Yaskawa INFORM job: tourneTRJ0.JBI

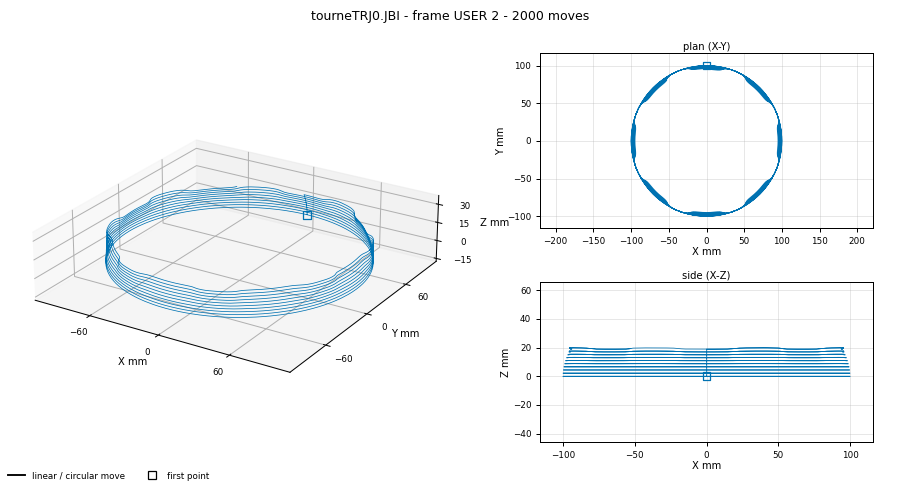
[picture p0: tool path of tourneTRJ0.JBI in frame USER 2, 2000 of 2000 moves have a stored position in this frame; points joined in program order, loops and branches not executed]
/JOB
//NAME tourneTRJ0
///FOLDERNAME DEMO
//POS
///NPOS 2000,0,2000,0,0,0
///USER 2
///TOOL 7
///POSTYPE USER
///RECTAN
///RCONF 1,0,0,0,0,0,0,0,0,0,0,0,0,0,0,0,0,0,0,0,0,0,0,0
C00000=0.000,100.000,0.000,-180.0000,-0.0000,-0.0000
C00001=5.792,99.832,0.000,-180.0000,0.0000,-3.3204
C00002=10.988,99.394,0.000,-180.0000,0.0000,-6.3084
C00003=15.564,98.781,0.000,-180.0000,0.0000,-8.9540
C00004=18.698,98.237,0.000,-180.0000,0.0000,-10.7765
C00005=20.854,97.801,0.000,-180.0000,0.0000,-12.0369
C00006=22.593,97.414,0.000,-180.0000,0.0000,-13.0576
C00007=24.351,96.990,0.000,-180.0000,0.0000,-14.0938
C00008=26.550,96.411,0.000,-180.0000,0.0000,-15.3967
C00009=29.248,95.627,0.000,-180.0000,0.0000,-17.0065
C00010=32.094,94.710,0.000,-180.0000,0.0000,-18.7198
C00011=34.739,93.772,0.000,-180.0000,0.0000,-20.3278
C00012=37.121,92.855,0.000,-180.0000,0.0000,-21.7902
C00013=39.410,91.907,0.000,-180.0000,0.0000,-23.2098
C00014=41.743,90.871,0.000,-180.0000,0.0000,-24.6724
C00015=44.276,89.664,0.000,180.0000,0.0000,-26.2801
C00016=46.937,88.300,0.000,180.0000,0.0000,-27.9935
C00017=49.400,86.946,0.000,-180.0000,0.0000,-29.6039
C00018=51.363,85.801,0.000,-180.0000,0.0000,-30.9060
C00019=52.906,84.858,0.000,-180.0000,0.0000,-31.9421
C00020=54.410,83.902,0.000,-180.0000,0.0000,-32.9632
C00021=56.242,82.685,0.000,-180.0000,0.0000,-34.2234
C00022=58.844,80.854,0.000,-180.0000,0.0000,-36.0464
C00023=62.512,78.053,0.000,-180.0000,0.0000,-38.6909
C00024=66.496,74.687,0.000,-180.0000,0.0000,-41.6796
C00025=70.711,70.711,0.000,-180.0000,0.0000,-45.0000
C00026=74.687,66.496,0.000,-180.0000,0.0000,-48.3204
C00027=78.053,62.512,0.000,-180.0000,0.0000,-51.3091
C00028=80.854,58.844,0.000,180.0000,0.0000,-53.9536
C00029=82.685,56.242,0.000,-180.0000,0.0000,-55.7766
C00030=83.902,54.410,0.000,-180.0000,0.0000,-57.0368
C00031=84.858,52.906,0.000,-180.0000,0.0000,-58.0579
C00032=85.801,51.363,0.000,-180.0000,0.0000,-59.0940
C00033=86.946,49.400,0.000,-180.0000,0.0000,-60.3961
C00034=88.300,46.937,0.000,-180.0000,0.0000,-62.0065
C00035=89.664,44.276,0.000,-180.0000,0.0000,-63.7199
C00036=90.871,41.743,0.000,-180.0000,0.0000,-65.3276
C00037=91.907,39.410,0.000,-180.0000,0.0000,-66.7902
C00038=92.855,37.121,0.000,-180.0000,0.0000,-68.2098
C00039=93.772,34.739,0.000,-180.0000,0.0000,-69.6722
C00040=94.710,32.094,0.000,-180.0000,0.0000,-71.2802
C00041=95.627,29.248,0.000,-180.0000,0.0000,-72.9935
C00042=96.411,26.550,0.000,-180.0000,0.0000,-74.6033
C00043=96.990,24.351,0.000,-180.0000,0.0000,-75.9062
C00044=97.414,22.593,0.000,-180.0000,0.0000,-76.9424
C00045=97.801,20.854,0.000,-180.0000,0.0000,-77.9631
C00046=98.237,18.698,0.000,-180.0000,0.0000,-79.2235
C00047=98.781,15.564,0.000,-180.0000,0.0000,-81.0460
C00048=99.394,10.988,0.000,-180.0000,0.0000,-83.6916
C00049=99.832,5.792,0.000,-180.0000,0.0000,-86.6796
C00050=100.000,0.000,0.000,-180.0000,0.0000,-90.0000
C00051=99.832,-5.792,0.000,-180.0000,0.0000,-93.3204
C00052=99.394,-10.988,0.000,-180.0000,0.0000,-96.3084
C00053=98.781,-15.564,0.000,-180.0000,0.0000,-98.9540
C00054=98.237,-18.698,0.000,-180.0000,0.0000,-100.7765
C00055=97.801,-20.854,0.000,-180.0000,0.0000,-102.0369
C00056=97.414,-22.593,0.000,-180.0000,0.0000,-103.0576
C00057=96.990,-24.351,0.000,-180.0000,0.0000,-104.0938
C00058=96.411,-26.550,0.000,-180.0000,0.0000,-105.3967
C00059=95.627,-29.248,0.000,-180.0000,0.0000,-107.0065
C00060=94.710,-32.094,0.000,-180.0000,0.0000,-108.7198
C00061=93.772,-34.739,0.000,-180.0000,0.0000,-110.3278
C00062=92.855,-37.121,0.000,-180.0000,0.0000,-111.7902
C00063=91.907,-39.410,0.000,-180.0000,0.0000,-113.2098
C00064=90.871,-41.743,0.000,-180.0000,0.0000,-114.6724
C00065=89.664,-44.276,0.000,-180.0000,0.0000,-116.2801
C00066=88.300,-46.937,0.000,-180.0000,0.0000,-117.9935
C00067=86.946,-49.400,0.000,-180.0000,0.0000,-119.6039
C00068=85.801,-51.363,0.000,-180.0000,0.0000,-120.9060
C00069=84.858,-52.906,0.000,-180.0000,0.0000,-121.9421
C00070=83.902,-54.410,0.000,-180.0000,0.0000,-122.9632
C00071=82.685,-56.242,0.000,-180.0000,0.0000,-124.2234
C00072=80.854,-58.844,0.000,-180.0000,0.0000,-126.0464
C00073=78.053,-62.512,0.000,-180.0000,0.0000,-128.6909
C00074=74.687,-66.496,0.000,-180.0000,0.0000,-131.6796
C00075=70.711,-70.711,0.000,-180.0000,0.0000,-135.0000
C00076=66.496,-74.687,0.000,-180.0000,0.0000,-138.3204
C00077=62.512,-78.053,0.000,-180.0000,0.0000,-141.3091
C00078=58.844,-80.854,0.000,-180.0000,0.0000,-143.9536
C00079=56.242,-82.685,0.000,-180.0000,0.0000,-145.7766
C00080=54.410,-83.902,0.000,-180.0000,0.0000,-147.0368
C00081=52.906,-84.858,0.000,-180.0000,0.0000,-148.0579
C00082=51.363,-85.801,0.000,-180.0000,0.0000,-149.0940
C00083=49.400,-86.946,0.000,180.0000,0.0000,-150.3961
C00084=46.937,-88.300,0.000,-180.0000,0.0000,-152.0065
C00085=44.276,-89.664,0.000,-180.0000,0.0000,-153.7199
C00086=41.743,-90.871,0.000,-180.0000,0.0000,-155.3276
C00087=39.410,-91.907,0.000,-180.0000,0.0000,-156.7902
C00088=37.121,-92.855,0.000,-180.0000,0.0000,-158.2098
C00089=34.739,-93.772,0.000,-180.0000,0.0000,-159.6722
C00090=32.094,-94.710,0.000,-180.0000,0.0000,-161.2802
C00091=29.248,-95.627,0.000,-180.0000,0.0000,-162.9935
C00092=26.550,-96.411,0.000,-180.0000,0.0000,-164.6033
C00093=24.351,-96.990,0.000,-180.0000,0.0000,-165.9062
C00094=22.593,-97.414,0.000,-180.0000,0.0000,-166.9424
C00095=20.854,-97.801,0.000,-180.0000,0.0000,-167.9631
C00096=18.698,-98.237,0.000,-180.0000,0.0000,-169.2235
C00097=15.564,-98.781,0.000,-180.0000,0.0000,-171.0460
C00098=10.988,-99.394,0.000,-180.0000,0.0000,-173.6916
C00099=5.792,-99.832,0.000,-180.0000,0.0000,-176.6796
C00100=0.000,-100.000,0.000,-180.0000,-0.0000,-180.0000
C00101=0.000,-100.000,0.000,-180.0000,-0.0000,-180.0000
C00102=-5.792,-99.832,0.000,180.0000,0.0000,-183.3204
C00103=-10.988,-99.394,0.000,180.0000,0.0000,-186.3084
C00104=-15.564,-98.781,0.000,180.0000,0.0000,-188.9540
C00105=-18.698,-98.237,0.000,180.0000,0.0000,-190.7765
C00106=-20.854,-97.801,0.000,180.0000,0.0000,-192.0369
C00107=-22.593,-97.414,0.000,180.0000,0.0000,-193.0576
C00108=-24.351,-96.990,0.000,180.0000,0.0000,-194.0938
C00109=-26.550,-96.411,0.000,180.0000,0.0000,-195.3967
C00110=-29.248,-95.627,0.000,180.0000,0.0000,-197.0065
C00111=-32.094,-94.710,0.000,180.0000,0.0000,-198.7198
C00112=-34.739,-93.772,0.000,180.0000,0.0000,-200.3278
C00113=-37.121,-92.855,0.000,180.0000,0.0000,-201.7902
C00114=-39.410,-91.907,0.000,180.0000,0.0000,-203.2098
C00115=-41.743,-90.871,0.000,180.0000,0.0000,-204.6724
C00116=-44.276,-89.664,0.000,180.0000,0.0000,-206.2801
C00117=-46.937,-88.300,0.000,180.0000,0.0000,-207.9935
C00118=-49.400,-86.946,0.000,180.0000,0.0000,-209.6039
C00119=-51.363,-85.801,0.000,180.0000,0.0000,-210.9060
C00120=-52.906,-84.858,0.000,180.0000,0.0000,-211.9421
C00121=-54.410,-83.902,0.000,180.0000,0.0000,-212.9632
C00122=-56.242,-82.685,0.000,180.0000,0.0000,-214.2234
C00123=-58.844,-80.854,0.000,180.0000,0.0000,-216.0464
C00124=-62.512,-78.053,0.000,180.0000,0.0000,-218.6909
C00125=-66.496,-74.687,0.000,180.0000,0.0000,-221.6796
C00126=-70.711,-70.711,0.000,180.0000,0.0000,-225.0000
C00127=-74.687,-66.496,0.000,180.0000,0.0000,-228.3204
C00128=-78.053,-62.512,0.000,180.0000,0.0000,-231.3091
C00129=-80.854,-58.844,0.000,180.0000,0.0000,-233.9536
C00130=-82.685,-56.242,0.000,180.0000,0.0000,-235.7766
C00131=-83.902,-54.410,0.000,180.0000,0.0000,-237.0368
C00132=-84.858,-52.906,0.000,180.0000,0.0000,-238.0579
C00133=-85.801,-51.363,0.000,180.0000,0.0000,-239.0940
C00134=-86.946,-49.400,0.000,180.0000,0.0000,-240.3961
C00135=-88.300,-46.937,0.000,180.0000,0.0000,-242.0065
C00136=-89.664,-44.276,0.000,180.0000,0.0000,-243.7199
C00137=-90.871,-41.743,0.000,-180.0000,0.0000,-245.3276
C00138=-91.907,-39.410,0.000,-180.0000,0.0000,-246.7902
C00139=-92.855,-37.121,0.000,180.0000,0.0000,-248.2098
C00140=-93.772,-34.739,0.000,180.0000,0.0000,-249.6722
C00141=-94.710,-32.094,0.000,-180.0000,0.0000,-251.2802
C00142=-95.627,-29.248,0.000,-180.0000,0.0000,-252.9935
C00143=-96.411,-26.550,0.000,180.0000,0.0000,-254.6033
C00144=-96.990,-24.351,0.000,180.0000,0.0000,-255.9062
C00145=-97.414,-22.593,0.000,180.0000,0.0000,-256.9424
C00146=-97.801,-20.854,0.000,180.0000,0.0000,-257.9631
C00147=-98.237,-18.698,0.000,180.0000,0.0000,-259.2235
C00148=-98.781,-15.564,0.000,180.0000,0.0000,-261.0460
C00149=-99.394,-10.988,0.000,180.0000,0.0000,-263.6916
C00150=-99.832,-5.792,0.000,180.0000,0.0000,-266.6796
C00151=-100.000,0.000,0.000,-180.0000,0.0000,-270.0000
C00152=-99.832,5.792,0.000,-180.0000,0.0000,-273.3204
C00153=-99.394,10.988,0.000,-180.0000,0.0000,-276.3084
C00154=-98.781,15.564,0.000,-180.0000,0.0000,-278.9540
C00155=-98.237,18.698,0.000,-180.0000,0.0000,-280.7765
C00156=-97.801,20.854,0.000,-180.0000,0.0000,-282.0369
C00157=-97.414,22.593,0.000,-180.0000,0.0000,-283.0576
C00158=-96.990,24.351,0.000,-180.0000,0.0000,-284.0938
C00159=-96.411,26.550,0.000,-180.0000,0.0000,-285.3967
C00160=-95.627,29.248,0.000,-180.0000,0.0000,-287.0065
C00161=-94.710,32.094,0.000,-180.0000,0.0000,-288.7198
C00162=-93.772,34.739,0.000,-180.0000,0.0000,-290.3278
C00163=-92.855,37.121,0.000,-180.0000,0.0000,-291.7902
C00164=-91.907,39.410,0.000,-180.0000,0.0000,-293.2098
C00165=-90.871,41.743,0.000,-180.0000,0.0000,-294.6724
C00166=-89.664,44.276,0.000,-180.0000,0.0000,-296.2801
C00167=-88.300,46.937,0.000,-180.0000,0.0000,-297.9935
C00168=-86.946,49.400,0.000,-180.0000,0.0000,-299.6039
C00169=-85.801,51.363,0.000,-180.0000,0.0000,-300.9060
C00170=-84.858,52.906,0.000,-180.0000,0.0000,-301.9421
C00171=-83.902,54.410,0.000,-180.0000,0.0000,-302.9632
C00172=-82.685,56.242,0.000,-180.0000,0.0000,-304.2234
C00173=-80.854,58.844,0.000,-180.0000,0.0000,-306.0464
C00174=-78.053,62.512,0.000,-180.0000,0.0000,-308.6909
C00175=-74.687,66.496,0.000,-180.0000,0.0000,-311.6796
C00176=-70.711,70.711,0.000,-180.0000,0.0000,-315.0000
C00177=-66.496,74.687,0.000,-180.0000,0.0000,-318.3204
C00178=-62.512,78.053,0.000,-180.0000,0.0000,-321.3091
C00179=-58.844,80.854,0.000,-180.0000,0.0000,-323.9536
C00180=-56.242,82.685,0.000,-180.0000,0.0000,-325.7766
C00181=-54.410,83.902,0.000,-180.0000,0.0000,-327.0368
C00182=-52.906,84.858,0.000,-180.0000,0.0000,-328.0579
C00183=-51.363,85.801,0.000,-180.0000,0.0000,-329.0940
C00184=-49.400,86.946,0.000,-180.0000,0.0000,-330.3961
C00185=-46.937,88.300,0.000,-180.0000,0.0000,-332.0065
C00186=-44.276,89.664,0.000,-180.0000,0.0000,-333.7199
C00187=-41.743,90.871,0.000,-180.0000,0.0000,-335.3276
C00188=-39.410,91.907,0.000,-180.0000,0.0000,-336.7902
C00189=-37.121,92.855,0.000,-180.0000,0.0000,-338.2098
C00190=-34.739,93.772,0.000,-180.0000,0.0000,-339.6722
C00191=-32.094,94.710,0.000,-180.0000,0.0000,-341.2802
C00192=-29.248,95.627,0.000,-180.0000,0.0000,-342.9935
C00193=-26.550,96.411,0.000,-180.0000,0.0000,-344.6033
C00194=-24.351,96.990,0.000,-180.0000,0.0000,-345.9062
C00195=-22.593,97.414,0.000,-180.0000,0.0000,-346.9424
C00196=-20.854,97.801,0.000,-180.0000,0.0000,-347.9631
C00197=-18.698,98.237,0.000,-180.0000,0.0000,-349.2235
C00198=-15.564,98.781,0.000,-180.0000,0.0000,-351.0460
C00199=-10.988,99.394,0.000,-180.0000,0.0000,-353.6916
C00200=-5.792,99.832,0.000,-180.0000,0.0000,-356.6796
C00201=0.000,100.000,0.000,-180.0000,0.0000,-360.0000
C00202=0.000,99.921,2.199,-175.9401,0.0000,-360.0000
C00203=5.785,99.754,2.199,-175.9390,-0.0000,-363.3190
C00204=10.976,99.317,2.199,-175.9440,0.0018,-366.3064
C00205=15.549,98.707,2.199,-176.1001,-0.0049,-368.9521
C00206=18.681,98.171,2.199,-176.5006,-0.0123,-370.7740
C00207=20.835,97.748,2.199,-177.0907,-0.0165,-372.0325
C00208=22.573,97.375,2.200,-177.7808,-0.0203,-373.0515
C00209=24.330,96.965,2.200,-178.4726,-0.0110,-374.0856
C00210=26.527,96.399,2.200,-179.0744,-0.0051,-375.3858
C00211=29.226,95.625,2.200,-179.5505,0.0004,-376.9948
C00212=32.077,94.713,2.200,-179.8732,-0.0006,-378.7100
C00213=34.728,93.776,2.200,-179.9819,-0.0006,-380.3211
C00214=37.118,92.856,2.200,-180.0000,0.0000,-381.7884
C00215=39.413,91.905,2.200,-180.0000,0.0000,-383.2118
C00216=41.753,90.866,2.200,-179.9796,0.0032,-384.6788
C00217=44.291,89.654,2.200,-179.8719,0.0006,-386.2904
C00218=46.951,88.283,2.200,-179.5514,0.0015,-388.0051
C00219=49.407,86.922,2.200,-179.0733,0.0071,-389.6142
C00220=51.360,85.768,2.200,-178.4728,0.0072,-390.9142
C00221=52.893,84.816,2.200,-177.7789,0.0198,-391.9485
C00222=54.385,83.851,2.199,-177.0907,0.0192,-392.9671
C00223=56.208,82.627,2.199,-176.5030,0.0134,-394.2260
C00224=58.802,80.791,2.199,-176.1018,0.0066,-396.0482
C00225=62.466,77.989,2.199,-175.9449,-0.0006,-398.6933
C00226=66.446,74.627,2.199,-175.9384,-0.0000,-401.6811
C00227=70.655,70.655,2.199,-175.9371,0.0000,-405.0000
C00228=74.627,66.446,2.199,-175.9384,0.0000,-408.3189
C00229=77.989,62.466,2.199,-175.9449,0.0006,-411.3067
C00230=80.791,58.802,2.199,-176.1018,-0.0066,-413.9518
C00231=82.627,56.208,2.199,-176.5030,-0.0134,-415.7740
C00232=83.851,54.385,2.199,-177.0907,-0.0192,-417.0329
C00233=84.816,52.893,2.200,-177.7789,-0.0198,-418.0515
C00234=85.768,51.360,2.200,-178.4728,-0.0072,-419.0858
C00235=86.922,49.407,2.200,-179.0733,-0.0071,-420.3858
C00236=88.283,46.951,2.200,-179.5514,-0.0015,-421.9949
C00237=89.654,44.291,2.200,-179.8719,-0.0006,-423.7096
C00238=90.866,41.753,2.200,-179.9796,-0.0032,-425.3212
C00239=91.905,39.413,2.200,-180.0000,0.0000,-426.7882
C00240=92.856,37.118,2.200,-180.0000,0.0000,-428.2116
C00241=93.776,34.728,2.200,-179.9819,0.0006,-429.6789
C00242=94.713,32.077,2.200,-179.8732,0.0006,-431.2900
C00243=95.625,29.226,2.200,-179.5505,-0.0004,-433.0052
C00244=96.399,26.527,2.200,-179.0744,0.0051,-434.6142
C00245=96.965,24.330,2.200,-178.4726,0.0110,-435.9144
C00246=97.375,22.573,2.200,-177.7808,0.0203,-436.9485
C00247=97.748,20.835,2.199,-177.0907,0.0165,-437.9675
C00248=98.171,18.681,2.199,-176.5006,0.0123,-439.2260
C00249=98.707,15.549,2.199,-176.1001,0.0049,-441.0479
C00250=99.317,10.976,2.199,-175.9440,-0.0018,-443.6936
C00251=99.754,5.785,2.199,-175.9390,0.0000,-446.6810
C00252=99.921,0.000,2.199,-175.9401,0.0000,-450.0000
C00253=99.754,-5.785,2.199,-175.9390,-0.0000,-453.3190
C00254=99.317,-10.976,2.199,-175.9440,0.0018,-456.3064
C00255=98.707,-15.549,2.199,-176.1001,-0.0049,-458.9521
C00256=98.171,-18.681,2.199,-176.5006,-0.0123,-460.7740
C00257=97.748,-20.835,2.199,-177.0907,-0.0165,-462.0325
C00258=97.375,-22.573,2.200,-177.7808,-0.0203,-463.0515
C00259=96.965,-24.330,2.200,-178.4726,-0.0110,-464.0856
C00260=96.399,-26.527,2.200,-179.0744,-0.0051,-465.3858
C00261=95.625,-29.226,2.200,-179.5505,0.0004,-466.9948
C00262=94.713,-32.077,2.200,-179.8732,-0.0006,-468.7100
C00263=93.776,-34.728,2.200,-179.9819,-0.0006,-470.3211
C00264=92.856,-37.118,2.200,-180.0000,0.0000,-471.7884
C00265=91.905,-39.413,2.200,-180.0000,0.0000,-473.2118
C00266=90.866,-41.753,2.200,-179.9796,0.0032,-474.6788
C00267=89.654,-44.291,2.200,-179.8719,0.0006,-476.2904
C00268=88.283,-46.951,2.200,-179.5514,0.0015,-478.0051
C00269=86.922,-49.407,2.200,-179.0733,0.0071,-479.6142
C00270=85.768,-51.360,2.200,-178.4728,0.0072,-480.9142
C00271=84.816,-52.893,2.200,-177.7789,0.0198,-481.9485
C00272=83.851,-54.385,2.199,-177.0907,0.0192,-482.9671
C00273=82.627,-56.208,2.199,-176.5030,0.0134,-484.2260
C00274=80.791,-58.802,2.199,-176.1018,0.0066,-486.0482
C00275=77.989,-62.466,2.199,-175.9449,-0.0006,-488.6933
C00276=74.627,-66.446,2.199,-175.9384,-0.0000,-491.6811
C00277=70.655,-70.655,2.199,-175.9371,-0.0000,-495.0000
C00278=66.446,-74.627,2.199,-175.9384,0.0000,-498.3189
C00279=62.466,-77.989,2.199,-175.9449,0.0006,-501.3067
C00280=58.802,-80.791,2.199,-176.1018,-0.0066,-503.9518
C00281=56.208,-82.627,2.199,-176.5030,-0.0134,-505.7740
C00282=54.385,-83.851,2.199,-177.0907,-0.0192,-507.0329
C00283=52.893,-84.816,2.200,-177.7789,-0.0198,-508.0515
C00284=51.360,-85.768,2.200,-178.4728,-0.0072,-509.0858
C00285=49.407,-86.922,2.200,-179.0733,-0.0071,-510.3858
C00286=46.951,-88.283,2.200,-179.5514,-0.0015,-511.9949
C00287=44.291,-89.654,2.200,-179.8719,-0.0006,-513.7096
C00288=41.753,-90.866,2.200,-179.9796,-0.0032,-515.3212
C00289=39.413,-91.905,2.200,-180.0000,0.0000,-516.7882
C00290=37.118,-92.856,2.200,-180.0000,0.0000,-518.2116
C00291=34.728,-93.776,2.200,-179.9819,0.0006,-519.6789
C00292=32.077,-94.713,2.200,-179.8732,0.0006,-521.2900
C00293=29.226,-95.625,2.200,-179.5505,-0.0004,-523.0052
C00294=26.527,-96.399,2.200,-179.0744,0.0051,-524.6142
C00295=24.330,-96.965,2.200,-178.4726,0.0110,-525.9144
C00296=22.573,-97.375,2.200,-177.7808,0.0203,-526.9485
C00297=20.835,-97.748,2.199,-177.0907,0.0165,-527.9675
C00298=18.681,-98.171,2.199,-176.5006,0.0123,-529.2260
C00299=15.549,-98.707,2.199,-176.1001,0.0049,-531.0479
C00300=10.976,-99.317,2.199,-175.9440,-0.0018,-533.6936
C00301=5.785,-99.754,2.199,-175.9390,0.0000,-536.6810
C00302=0.000,-99.921,2.199,-175.9401,0.0000,-540.0000
C00303=0.000,-99.921,2.199,-175.9401,0.0000,-540.0000
C00304=-5.785,-99.754,2.199,-175.9390,-0.0000,-543.3190
C00305=-10.976,-99.317,2.199,-175.9440,0.0018,-546.3064
C00306=-15.549,-98.707,2.199,-176.1001,-0.0049,-548.9521
C00307=-18.681,-98.171,2.199,-176.5006,-0.0123,-550.7740
C00308=-20.835,-97.748,2.199,-177.0907,-0.0165,-552.0325
C00309=-22.573,-97.375,2.200,-177.7808,-0.0203,-553.0515
C00310=-24.330,-96.965,2.200,-178.4726,-0.0110,-554.0856
C00311=-26.527,-96.399,2.200,-179.0744,-0.0051,-555.3858
C00312=-29.226,-95.625,2.200,-179.5505,0.0004,-556.9948
C00313=-32.077,-94.713,2.200,-179.8732,-0.0006,-558.7100
C00314=-34.728,-93.776,2.200,-179.9819,-0.0006,-560.3211
C00315=-37.118,-92.856,2.200,-180.0000,0.0000,-561.7884
C00316=-39.413,-91.905,2.200,-180.0000,0.0000,-563.2118
C00317=-41.753,-90.866,2.200,-179.9796,0.0032,-564.6788
C00318=-44.291,-89.654,2.200,-179.8719,0.0006,-566.2904
C00319=-46.951,-88.283,2.200,-179.5514,0.0015,-568.0051
C00320=-49.407,-86.922,2.200,-179.0733,0.0071,-569.6142
C00321=-51.360,-85.768,2.200,-178.4728,0.0072,-570.9142
C00322=-52.893,-84.816,2.200,-177.7789,0.0198,-571.9485
C00323=-54.385,-83.851,2.199,-177.0907,0.0192,-572.9671
C00324=-56.208,-82.627,2.199,-176.5030,0.0134,-574.2260
C00325=-58.802,-80.791,2.199,-176.1018,0.0066,-576.0482
C00326=-62.466,-77.989,2.199,-175.9449,-0.0006,-578.6933
C00327=-66.446,-74.627,2.199,-175.9384,-0.0000,-581.6811
C00328=-70.655,-70.655,2.199,-175.9371,-0.0000,-585.0000
C00329=-74.627,-66.446,2.199,-175.9384,0.0000,-588.3189
C00330=-77.989,-62.466,2.199,-175.9449,0.0006,-591.3067
C00331=-80.791,-58.802,2.199,-176.1018,-0.0066,-593.9518
C00332=-82.627,-56.208,2.199,-176.5030,-0.0134,-595.7740
C00333=-83.851,-54.385,2.199,-177.0907,-0.0192,-597.0329
C00334=-84.816,-52.893,2.200,-177.7789,-0.0198,-598.0515
C00335=-85.768,-51.360,2.200,-178.4728,-0.0072,-599.0858
C00336=-86.922,-49.407,2.200,-179.0733,-0.0071,-600.3858
C00337=-88.283,-46.951,2.200,-179.5514,-0.0015,-601.9949
C00338=-89.654,-44.291,2.200,-179.8719,-0.0006,-603.7096
C00339=-90.866,-41.753,2.200,-179.9796,-0.0032,-605.3212
C00340=-91.905,-39.413,2.200,-180.0000,0.0000,-606.7882
C00341=-92.856,-37.118,2.200,-180.0000,0.0000,-608.2116
C00342=-93.776,-34.728,2.200,-179.9819,0.0006,-609.6789
C00343=-94.713,-32.077,2.200,-179.8732,0.0006,-611.2900
C00344=-95.625,-29.226,2.200,-179.5505,-0.0004,-613.0052
C00345=-96.399,-26.527,2.200,-179.0744,0.0051,-614.6142
C00346=-96.965,-24.330,2.200,-178.4726,0.0110,-615.9144
C00347=-97.375,-22.573,2.200,-177.7808,0.0203,-616.9485
C00348=-97.748,-20.835,2.199,-177.0907,0.0165,-617.9675
C00349=-98.171,-18.681,2.199,-176.5006,0.0123,-619.2260
C00350=-98.707,-15.549,2.199,-176.1001,0.0049,-621.0479
C00351=-99.317,-10.976,2.199,-175.9440,-0.0018,-623.6936
C00352=-99.754,-5.785,2.199,-175.9390,0.0000,-626.6810
C00353=-99.921,0.000,2.199,-175.9401,0.0000,-630.0000
C00354=-99.754,5.785,2.199,-175.9390,-0.0000,-633.3190
C00355=-99.317,10.976,2.199,-175.9440,0.0018,-636.3064
C00356=-98.707,15.549,2.199,-176.1001,-0.0049,-638.9521
C00357=-98.171,18.681,2.199,-176.5006,-0.0123,-640.7740
C00358=-97.748,20.835,2.199,-177.0907,-0.0165,-642.0325
C00359=-97.375,22.573,2.200,-177.7808,-0.0203,-643.0515
C00360=-96.965,24.330,2.200,-178.4726,-0.0110,-644.0856
C00361=-96.399,26.527,2.200,-179.0744,-0.0051,-645.3858
C00362=-95.625,29.226,2.200,-179.5505,0.0004,-646.9948
C00363=-94.713,32.077,2.200,-179.8732,-0.0006,-648.7100
C00364=-93.776,34.728,2.200,-179.9819,-0.0006,-650.3211
C00365=-92.856,37.118,2.200,-180.0000,0.0000,-651.7884
C00366=-91.905,39.413,2.200,-180.0000,0.0000,-653.2118
C00367=-90.866,41.753,2.200,-179.9796,0.0032,-654.6788
C00368=-89.654,44.291,2.200,-179.8719,0.0006,-656.2904
C00369=-88.283,46.951,2.200,-179.5514,0.0015,-658.0051
C00370=-86.922,49.407,2.200,-179.0733,0.0071,-659.6142
C00371=-85.768,51.360,2.200,-178.4728,0.0072,-660.9142
C00372=-84.816,52.893,2.200,-177.7789,0.0198,-661.9485
C00373=-83.851,54.385,2.199,-177.0907,0.0192,-662.9671
C00374=-82.627,56.208,2.199,-176.5030,0.0134,-664.2260
C00375=-80.791,58.802,2.199,-176.1018,0.0066,-666.0482
C00376=-77.989,62.466,2.199,-175.9449,-0.0006,-668.6933
C00377=-74.627,66.446,2.199,-175.9384,-0.0000,-671.6811
C00378=-70.655,70.655,2.199,-175.9371,-0.0000,-675.0000
C00379=-66.446,74.627,2.199,-175.9384,0.0000,-678.3189
C00380=-62.466,77.989,2.199,-175.9449,0.0006,-681.3067
C00381=-58.802,80.791,2.199,-176.1018,-0.0066,-683.9518
C00382=-56.208,82.627,2.199,-176.5030,-0.0134,-685.7740
C00383=-54.385,83.851,2.199,-177.0907,-0.0192,-687.0329
C00384=-52.893,84.816,2.200,-177.7789,-0.0198,-688.0515
C00385=-51.360,85.768,2.200,-178.4728,-0.0072,-689.0858
C00386=-49.407,86.922,2.200,-179.0733,-0.0071,-690.3858
C00387=-46.951,88.283,2.200,-179.5514,-0.0015,-691.9949
C00388=-44.291,89.654,2.200,-179.8719,-0.0006,-693.7096
C00389=-41.753,90.866,2.200,-179.9796,-0.0032,-695.3212
C00390=-39.413,91.905,2.200,-180.0000,0.0000,-696.7882
C00391=-37.118,92.856,2.200,-180.0000,0.0000,-698.2116
C00392=-34.728,93.776,2.200,-179.9819,0.0006,-699.6789
C00393=-32.077,94.713,2.200,-179.8732,0.0006,-701.2900
C00394=-29.226,95.625,2.200,-179.5505,-0.0004,-703.0052
C00395=-26.527,96.399,2.200,-179.0744,0.0051,-704.6142
C00396=-24.330,96.965,2.200,-178.4726,0.0110,-705.9144
C00397=-22.573,97.375,2.200,-177.7808,0.0203,-706.9485
C00398=-20.835,97.748,2.199,-177.0907,0.0165,-707.9675
C00399=-18.681,98.171,2.199,-176.5006,0.0123,-709.2260
C00400=-15.549,98.707,2.199,-176.1001,0.0049,-711.0479
C00401=-10.976,99.317,2.199,-175.9440,-0.0018,-713.6936
C00402=-5.785,99.754,2.199,-175.9390,0.0000,-716.6810
C00403=0.000,99.921,2.199,-175.9401,0.0000,-720.0000
C00404=0.000,99.691,4.387,-172.1025,0.0000,-720.0000
C00405=5.764,99.524,4.387,-172.1006,0.0031,-723.3146
C00406=10.941,99.090,4.387,-172.1132,-0.0092,-726.3008
C00407=15.506,98.490,4.388,-172.4149,-0.0426,-728.9471
C00408=18.630,97.979,4.390,-173.1917,-0.1025,-730.7659
C00409=20.779,97.591,4.393,-174.3456,-0.1482,-732.0199
C00410=22.514,97.259,4.396,-175.6935,-0.1377,-733.0335
C00411=24.268,96.890,4.398,-177.0472,-0.0778,-734.0616
C00412=26.460,96.362,4.399,-178.2128,-0.0272,-735.3544
C00413=29.164,95.617,4.399,-179.1461,-0.0089,-736.9622
C00414=32.027,94.722,4.399,-179.7590,-0.0028,-738.6812
C00415=34.697,93.786,4.400,-179.9638,-0.0012,-740.3024
C00416=37.107,92.860,4.400,-179.9947,-0.0021,-741.7817
C00417=39.424,91.901,4.400,-179.9947,-0.0023,-743.2185
C00418=41.782,90.851,4.400,-179.9616,0.0013,-744.6975
C00419=44.332,89.625,4.399,-179.7566,0.0010,-746.3188
C00420=46.990,88.233,4.399,-179.1436,0.0113,-748.0383
C00421=49.428,86.848,4.399,-178.2096,0.0294,-749.6456
C00422=51.352,85.672,4.398,-177.0480,0.0751,-750.9386
C00423=52.853,84.692,4.396,-175.6950,0.1393,-751.9667
C00424=54.314,83.700,4.393,-174.3428,0.1470,-752.9801
C00425=56.108,82.455,4.390,-173.1912,0.1047,-754.2340
C00426=58.679,80.608,4.388,-172.4131,0.0429,-756.0529
C00427=62.331,77.804,4.387,-172.1130,0.0081,-758.6992
C00428=66.299,74.450,4.387,-172.0978,-0.0024,-761.6856
C00429=70.493,70.493,4.387,-172.0990,-0.0000,-765.0000
C00430=74.450,66.299,4.387,-172.0978,0.0024,-768.3144
C00431=77.804,62.331,4.387,-172.1130,-0.0081,-771.3008
C00432=80.608,58.679,4.388,-172.4131,-0.0429,-773.9471
C00433=82.455,56.108,4.390,-173.1912,-0.1047,-775.7660
C00434=83.700,54.314,4.393,-174.3428,-0.1470,-777.0199
C00435=84.692,52.853,4.396,-175.6950,-0.1393,-778.0333
C00436=85.672,51.352,4.398,-177.0480,-0.0751,-779.0614
C00437=86.848,49.428,4.399,-178.2096,-0.0294,-780.3544
C00438=88.233,46.990,4.399,-179.1436,-0.0113,-781.9617
C00439=89.625,44.332,4.399,-179.7566,-0.0010,-783.6812
C00440=90.851,41.782,4.400,-179.9616,-0.0013,-785.3025
C00441=91.901,39.424,4.400,-179.9947,0.0023,-786.7815
C00442=92.860,37.107,4.400,-179.9947,0.0021,-788.2183
C00443=93.786,34.697,4.400,-179.9638,0.0012,-789.6976
C00444=94.722,32.027,4.399,-179.7590,0.0028,-791.3188
C00445=95.617,29.164,4.399,-179.1461,0.0089,-793.0378
C00446=96.362,26.460,4.399,-178.2128,0.0272,-794.6456
C00447=96.890,24.268,4.398,-177.0472,0.0778,-795.9384
C00448=97.259,22.514,4.396,-175.6935,0.1377,-796.9665
C00449=97.591,20.779,4.393,-174.3456,0.1482,-797.9801
C00450=97.979,18.630,4.390,-173.1917,0.1025,-799.2341
C00451=98.490,15.506,4.388,-172.4149,0.0426,-801.0529
C00452=99.090,10.941,4.387,-172.1132,0.0092,-803.6992
C00453=99.524,5.764,4.387,-172.1006,-0.0031,-806.6854
C00454=99.691,0.000,4.387,-172.1025,0.0000,-810.0000
C00455=99.524,-5.764,4.387,-172.1006,0.0031,-813.3146
C00456=99.090,-10.941,4.387,-172.1132,-0.0092,-816.3008
C00457=98.490,-15.506,4.388,-172.4149,-0.0426,-818.9471
C00458=97.979,-18.630,4.390,-173.1917,-0.1025,-820.7659
C00459=97.591,-20.779,4.393,-174.3456,-0.1482,-822.0199
C00460=97.259,-22.514,4.396,-175.6935,-0.1377,-823.0335
C00461=96.890,-24.268,4.398,-177.0472,-0.0778,-824.0616
C00462=96.362,-26.460,4.399,-178.2128,-0.0272,-825.3544
C00463=95.617,-29.164,4.399,-179.1461,-0.0089,-826.9622
C00464=94.722,-32.027,4.399,-179.7590,-0.0028,-828.6812
C00465=93.786,-34.697,4.400,-179.9638,-0.0012,-830.3024
C00466=92.860,-37.107,4.400,-179.9947,-0.0021,-831.7817
C00467=91.901,-39.424,4.400,-179.9947,-0.0023,-833.2185
C00468=90.851,-41.782,4.400,-179.9616,0.0013,-834.6975
C00469=89.625,-44.332,4.399,-179.7566,0.0010,-836.3188
C00470=88.233,-46.990,4.399,-179.1436,0.0113,-838.0383
C00471=86.848,-49.428,4.399,-178.2096,0.0294,-839.6456
C00472=85.672,-51.352,4.398,-177.0480,0.0751,-840.9386
C00473=84.692,-52.853,4.396,-175.6950,0.1393,-841.9667
C00474=83.700,-54.314,4.393,-174.3428,0.1470,-842.9801
C00475=82.455,-56.108,4.390,-173.1912,0.1047,-844.2340
C00476=80.608,-58.679,4.388,-172.4131,0.0429,-846.0529
C00477=77.804,-62.331,4.387,-172.1130,0.0081,-848.6992
C00478=74.450,-66.299,4.387,-172.0978,-0.0024,-851.6856
C00479=70.493,-70.493,4.387,-172.0990,-0.0000,-855.0000
C00480=66.299,-74.450,4.387,-172.0978,0.0024,-858.3144
C00481=62.331,-77.804,4.387,-172.1130,-0.0081,-861.3008
C00482=58.679,-80.608,4.388,-172.4131,-0.0429,-863.9471
C00483=56.108,-82.455,4.390,-173.1912,-0.1047,-865.7660
C00484=54.314,-83.700,4.393,-174.3428,-0.1470,-867.0199
C00485=52.853,-84.692,4.396,-175.6950,-0.1393,-868.0333
C00486=51.352,-85.672,4.398,-177.0480,-0.0751,-869.0614
C00487=49.428,-86.848,4.399,-178.2096,-0.0294,-870.3544
C00488=46.990,-88.233,4.399,-179.1436,-0.0113,-871.9617
C00489=44.332,-89.625,4.399,-179.7566,-0.0010,-873.6812
C00490=41.782,-90.851,4.400,-179.9616,-0.0013,-875.3025
C00491=39.424,-91.901,4.400,-179.9947,0.0023,-876.7815
C00492=37.107,-92.860,4.400,-179.9947,0.0021,-878.2183
C00493=34.697,-93.786,4.400,-179.9638,0.0012,-879.6976
C00494=32.027,-94.722,4.399,-179.7590,0.0028,-881.3188
C00495=29.164,-95.617,4.399,-179.1461,0.0089,-883.0378
C00496=26.460,-96.362,4.399,-178.2128,0.0272,-884.6456
C00497=24.268,-96.890,4.398,-177.0472,0.0778,-885.9384
C00498=22.514,-97.259,4.396,-175.6935,0.1377,-886.9665
C00499=20.779,-97.591,4.393,-174.3456,0.1482,-887.9801
C00500=18.630,-97.979,4.390,-173.1917,0.1025,-889.2341
C00501=15.506,-98.490,4.388,-172.4149,0.0426,-891.0529
C00502=10.941,-99.090,4.387,-172.1132,0.0092,-893.6992
C00503=5.764,-99.524,4.387,-172.1006,-0.0031,-896.6854
C00504=0.000,-99.691,4.387,-172.1025,0.0000,-900.0000
C00505=0.000,-99.691,4.387,-172.1025,0.0000,-900.0000
C00506=-5.764,-99.524,4.387,-172.1006,0.0031,-903.3146
C00507=-10.941,-99.090,4.387,-172.1132,-0.0092,-906.3008
C00508=-15.506,-98.490,4.388,-172.4149,-0.0426,-908.9471
C00509=-18.630,-97.979,4.390,-173.1917,-0.1025,-910.7659
C00510=-20.779,-97.591,4.393,-174.3456,-0.1482,-912.0199
C00511=-22.514,-97.259,4.396,-175.6935,-0.1377,-913.0335
C00512=-24.268,-96.890,4.398,-177.0472,-0.0778,-914.0616
C00513=-26.460,-96.362,4.399,-178.2128,-0.0272,-915.3544
C00514=-29.164,-95.617,4.399,-179.1461,-0.0089,-916.9622
C00515=-32.027,-94.722,4.399,-179.7590,-0.0028,-918.6812
C00516=-34.697,-93.786,4.400,-179.9638,-0.0012,-920.3024
C00517=-37.107,-92.860,4.400,-179.9947,-0.0021,-921.7817
C00518=-39.424,-91.901,4.400,-179.9947,-0.0023,-923.2185
C00519=-41.782,-90.851,4.400,-179.9616,0.0013,-924.6975
C00520=-44.332,-89.625,4.399,-179.7566,0.0010,-926.3188
C00521=-46.990,-88.233,4.399,-179.1436,0.0113,-928.0383
C00522=-49.428,-86.848,4.399,-178.2096,0.0294,-929.6456
C00523=-51.352,-85.672,4.398,-177.0480,0.0751,-930.9386
C00524=-52.853,-84.692,4.396,-175.6950,0.1393,-931.9667
C00525=-54.314,-83.700,4.393,-174.3428,0.1470,-932.9801
C00526=-56.108,-82.455,4.390,-173.1912,0.1047,-934.2340
C00527=-58.679,-80.608,4.388,-172.4131,0.0429,-936.0529
C00528=-62.331,-77.804,4.387,-172.1130,0.0081,-938.6992
C00529=-66.299,-74.450,4.387,-172.0978,-0.0024,-941.6856
C00530=-70.493,-70.493,4.387,-172.0990,-0.0000,-945.0000
C00531=-74.450,-66.299,4.387,-172.0978,0.0024,-948.3144
C00532=-77.804,-62.331,4.387,-172.1130,-0.0081,-951.3008
C00533=-80.608,-58.679,4.388,-172.4131,-0.0429,-953.9471
C00534=-82.455,-56.108,4.390,-173.1912,-0.1047,-955.7660
C00535=-83.700,-54.314,4.393,-174.3428,-0.1470,-957.0199
C00536=-84.692,-52.853,4.396,-175.6950,-0.1393,-958.0333
C00537=-85.672,-51.352,4.398,-177.0480,-0.0751,-959.0614
C00538=-86.848,-49.428,4.399,-178.2096,-0.0294,-960.3544
C00539=-88.233,-46.990,4.399,-179.1436,-0.0113,-961.9617
C00540=-89.625,-44.332,4.399,-179.7566,-0.0010,-963.6812
C00541=-90.851,-41.782,4.400,-179.9616,-0.0013,-965.3025
C00542=-91.901,-39.424,4.400,-179.9947,0.0023,-966.7815
C00543=-92.860,-37.107,4.400,-179.9947,0.0021,-968.2183
C00544=-93.786,-34.697,4.400,-179.9638,0.0012,-969.6976
C00545=-94.722,-32.027,4.399,-179.7590,0.0028,-971.3188
C00546=-95.617,-29.164,4.399,-179.1461,0.0089,-973.0378
C00547=-96.362,-26.460,4.399,-178.2128,0.0272,-974.6456
C00548=-96.890,-24.268,4.398,-177.0472,0.0778,-975.9384
C00549=-97.259,-22.514,4.396,-175.6935,0.1377,-976.9665
C00550=-97.591,-20.779,4.393,-174.3456,0.1482,-977.9801
C00551=-97.979,-18.630,4.390,-173.1917,0.1025,-979.2341
C00552=-98.490,-15.506,4.388,-172.4149,0.0426,-981.0529
C00553=-99.090,-10.941,4.387,-172.1132,0.0092,-983.6992
C00554=-99.524,-5.764,4.387,-172.1006,-0.0031,-986.6854
C00555=-99.691,0.000,4.387,-172.1025,-0.0000,-990.0000
C00556=-99.524,5.764,4.387,-172.1006,0.0031,-993.3146
C00557=-99.090,10.941,4.387,-172.1132,-0.0092,-996.3008
C00558=-98.490,15.506,4.388,-172.4149,-0.0426,-998.9471
C00559=-97.979,18.630,4.390,-173.1917,-0.1025,-1000.7659
C00560=-97.591,20.779,4.393,-174.3456,-0.1482,-1002.0199
C00561=-97.259,22.514,4.396,-175.6935,-0.1377,-1003.0335
C00562=-96.890,24.268,4.398,-177.0472,-0.0778,-1004.0616
C00563=-96.362,26.460,4.399,-178.2128,-0.0272,-1005.3544
C00564=-95.617,29.164,4.399,-179.1461,-0.0089,-1006.9622
C00565=-94.722,32.027,4.399,-179.7590,-0.0028,-1008.6812
C00566=-93.786,34.697,4.400,-179.9638,-0.0012,-1010.3024
C00567=-92.860,37.107,4.400,-179.9947,-0.0021,-1011.7817
C00568=-91.901,39.424,4.400,-179.9947,-0.0023,-1013.2185
C00569=-90.851,41.782,4.400,-179.9616,0.0013,-1014.6975
C00570=-89.625,44.332,4.399,-179.7566,0.0010,-1016.3188
C00571=-88.233,46.990,4.399,-179.1436,0.0113,-1018.0383
C00572=-86.848,49.428,4.399,-178.2096,0.0294,-1019.6456
C00573=-85.672,51.352,4.398,-177.0480,0.0751,-1020.9386
C00574=-84.692,52.853,4.396,-175.6950,0.1393,-1021.9667
C00575=-83.700,54.314,4.393,-174.3428,0.1470,-1022.9801
C00576=-82.455,56.108,4.390,-173.1912,0.1047,-1024.2340
C00577=-80.608,58.679,4.388,-172.4131,0.0429,-1026.0529
C00578=-77.804,62.331,4.387,-172.1130,0.0081,-1028.6992
C00579=-74.450,66.299,4.387,-172.0978,-0.0024,-1031.6856
C00580=-70.493,70.493,4.387,-172.0990,0.0000,-1035.0000
C00581=-66.299,74.450,4.387,-172.0978,0.0024,-1038.3144
C00582=-62.331,77.804,4.387,-172.1130,-0.0081,-1041.3008
C00583=-58.679,80.608,4.388,-172.4131,-0.0429,-1043.9471
C00584=-56.108,82.455,4.390,-173.1912,-0.1047,-1045.7660
C00585=-54.314,83.700,4.393,-174.3428,-0.1470,-1047.0199
C00586=-52.853,84.692,4.396,-175.6950,-0.1393,-1048.0333
C00587=-51.352,85.672,4.398,-177.0480,-0.0751,-1049.0614
C00588=-49.428,86.848,4.399,-178.2096,-0.0294,-1050.3544
C00589=-46.990,88.233,4.399,-179.1436,-0.0113,-1051.9617
C00590=-44.332,89.625,4.399,-179.7566,-0.0010,-1053.6812
C00591=-41.782,90.851,4.400,-179.9616,-0.0013,-1055.3025
C00592=-39.424,91.901,4.400,-179.9947,0.0023,-1056.7815
C00593=-37.107,92.860,4.400,-179.9947,0.0021,-1058.2183
C00594=-34.697,93.786,4.400,-179.9638,0.0012,-1059.6976
C00595=-32.027,94.722,4.399,-179.7590,0.0028,-1061.3188
C00596=-29.164,95.617,4.399,-179.1461,0.0089,-1063.0378
C00597=-26.460,96.362,4.399,-178.2128,0.0272,-1064.6456
C00598=-24.268,96.890,4.398,-177.0472,0.0778,-1065.9384
C00599=-22.514,97.259,4.396,-175.6935,0.1377,-1066.9665
C00600=-20.779,97.591,4.393,-174.3456,0.1482,-1067.9801
C00601=-18.630,97.979,4.390,-173.1917,0.1025,-1069.2341
C00602=-15.506,98.490,4.388,-172.4149,0.0426,-1071.0529
C00603=-10.941,99.090,4.387,-172.1132,0.0092,-1073.6992
C00604=-5.764,99.524,4.387,-172.1006,-0.0031,-1076.6854
C00605=0.000,99.691,4.387,-172.1025,0.0000,-1080.0000
C00606=0.000,99.321,6.555,-168.5271,0.0000,-1080.0000
C00607=5.730,99.155,6.555,-168.5253,0.0014,-1083.3073
C00608=10.884,98.723,6.555,-168.5476,-0.0211,-1086.2913
C00609=15.437,98.140,6.558,-168.9780,-0.1303,-1088.9391
C00610=18.547,97.668,6.566,-170.1170,-0.3386,-1090.7524
C00611=20.687,97.336,6.576,-171.8150,-0.4851,-1091.9986
C00612=22.417,97.071,6.585,-173.8031,-0.4429,-1093.0036
C00613=24.167,96.770,6.592,-175.7648,-0.2484,-1094.0220
C00614=26.351,96.303,6.595,-177.4464,-0.0927,-1095.3030
C00615=29.062,95.605,6.597,-178.7866,-0.0275,-1096.9082
C00616=31.947,94.737,6.598,-179.6630,-0.0048,-1098.6350
C00617=34.646,93.803,6.599,-179.9457,-0.0017,-1100.2716
C00618=37.090,92.867,6.600,-179.9947,-0.0021,-1101.7712
C00619=39.440,91.893,6.600,-179.9947,-0.0023,-1103.2288
C00620=41.830,90.827,6.599,-179.9436,-0.0008,-1104.7282
C00621=44.399,89.579,6.598,-179.6644,0.0063,-1106.3649
C00622=47.053,88.152,6.597,-178.7893,0.0293,-1108.0920
C00623=49.464,86.729,6.595,-177.4408,0.0910,-1109.6973
C00624=51.338,85.515,6.592,-175.7651,0.2472,-1110.9780
C00625=52.788,84.491,6.585,-173.8020,0.4415,-1111.9962
C00626=54.199,83.455,6.576,-171.8109,0.4845,-1113.0013
C00627=55.947,82.176,6.566,-170.1166,0.3384,-1114.2478
C00628=58.480,80.311,6.558,-168.9774,0.1342,-1116.0610
C00629=62.112,77.504,6.555,-168.5500,0.0193,-1118.7088
C00630=66.061,74.165,6.555,-168.5237,-0.0027,-1121.6924
C00631=70.230,70.230,6.555,-168.5306,-0.0000,-1125.0000
C00632=74.165,66.061,6.555,-168.5237,0.0027,-1128.3076
C00633=77.504,62.112,6.555,-168.5500,-0.0193,-1131.2912
C00634=80.311,58.480,6.558,-168.9774,-0.1342,-1133.9390
C00635=82.176,55.947,6.566,-170.1166,-0.3384,-1135.7522
C00636=83.455,54.199,6.576,-171.8109,-0.4845,-1136.9987
C00637=84.491,52.788,6.585,-173.8020,-0.4415,-1138.0038
C00638=85.515,51.338,6.592,-175.7651,-0.2472,-1139.0220
C00639=86.729,49.464,6.595,-177.4408,-0.0910,-1140.3027
C00640=88.152,47.053,6.597,-178.7893,-0.0293,-1141.9080
C00641=89.579,44.399,6.598,-179.6644,-0.0063,-1143.6351
C00642=90.827,41.830,6.599,-179.9436,0.0008,-1145.2718
C00643=91.893,39.440,6.600,-179.9947,0.0023,-1146.7712
C00644=92.867,37.090,6.600,-179.9947,0.0021,-1148.2288
C00645=93.803,34.646,6.599,-179.9457,0.0017,-1149.7284
C00646=94.737,31.947,6.598,-179.6630,0.0048,-1151.3650
C00647=95.605,29.062,6.597,-178.7866,0.0275,-1153.0918
C00648=96.303,26.351,6.595,-177.4464,0.0927,-1154.6970
C00649=96.770,24.167,6.592,-175.7648,0.2484,-1155.9780
C00650=97.071,22.417,6.585,-173.8031,0.4429,-1156.9964
C00651=97.336,20.687,6.576,-171.8150,0.4851,-1158.0014
C00652=97.668,18.547,6.566,-170.1170,0.3386,-1159.2476
C00653=98.140,15.437,6.558,-168.9780,0.1303,-1161.0609
C00654=98.723,10.884,6.555,-168.5476,0.0211,-1163.7087
C00655=99.155,5.730,6.555,-168.5253,-0.0014,-1166.6927
C00656=99.321,0.000,6.555,-168.5271,-0.0000,-1170.0000
C00657=99.155,-5.730,6.555,-168.5253,0.0014,-1173.3073
C00658=98.723,-10.884,6.555,-168.5476,-0.0211,-1176.2913
C00659=98.140,-15.437,6.558,-168.9780,-0.1303,-1178.9391
C00660=97.668,-18.547,6.566,-170.1170,-0.3386,-1180.7524
C00661=97.336,-20.687,6.576,-171.8150,-0.4851,-1181.9986
C00662=97.071,-22.417,6.585,-173.8031,-0.4429,-1183.0036
C00663=96.770,-24.167,6.592,-175.7648,-0.2484,-1184.0220
C00664=96.303,-26.351,6.595,-177.4464,-0.0927,-1185.3030
C00665=95.605,-29.062,6.597,-178.7866,-0.0275,-1186.9082
C00666=94.737,-31.947,6.598,-179.6630,-0.0048,-1188.6350
C00667=93.803,-34.646,6.599,-179.9457,-0.0017,-1190.2716
C00668=92.867,-37.090,6.600,-179.9947,-0.0021,-1191.7712
C00669=91.893,-39.440,6.600,-179.9947,-0.0023,-1193.2288
C00670=90.827,-41.830,6.599,-179.9436,-0.0008,-1194.7282
C00671=89.579,-44.399,6.598,-179.6644,0.0063,-1196.3649
C00672=88.152,-47.053,6.597,-178.7893,0.0293,-1198.0920
C00673=86.729,-49.464,6.595,-177.4408,0.0910,-1199.6973
C00674=85.515,-51.338,6.592,-175.7651,0.2472,-1200.9780
C00675=84.491,-52.788,6.585,-173.8020,0.4415,-1201.9962
C00676=83.455,-54.199,6.576,-171.8109,0.4845,-1203.0013
C00677=82.176,-55.947,6.566,-170.1166,0.3384,-1204.2478
C00678=80.311,-58.480,6.558,-168.9774,0.1342,-1206.0610
C00679=77.504,-62.112,6.555,-168.5500,0.0193,-1208.7088
C00680=74.165,-66.061,6.555,-168.5237,-0.0027,-1211.6924
C00681=70.230,-70.230,6.555,-168.5306,0.0000,-1215.0000
C00682=66.061,-74.165,6.555,-168.5237,0.0027,-1218.3076
C00683=62.112,-77.504,6.555,-168.5500,-0.0193,-1221.2912
C00684=58.480,-80.311,6.558,-168.9774,-0.1342,-1223.9390
C00685=55.947,-82.176,6.566,-170.1166,-0.3384,-1225.7522
C00686=54.199,-83.455,6.576,-171.8109,-0.4845,-1226.9987
C00687=52.788,-84.491,6.585,-173.8020,-0.4415,-1228.0038
C00688=51.338,-85.515,6.592,-175.7651,-0.2472,-1229.0220
C00689=49.464,-86.729,6.595,-177.4408,-0.0910,-1230.3027
C00690=47.053,-88.152,6.597,-178.7893,-0.0293,-1231.9080
C00691=44.399,-89.579,6.598,-179.6644,-0.0063,-1233.6351
C00692=41.830,-90.827,6.599,-179.9436,0.0008,-1235.2718
C00693=39.440,-91.893,6.600,-179.9947,0.0023,-1236.7712
C00694=37.090,-92.867,6.600,-179.9947,0.0021,-1238.2288
C00695=34.646,-93.803,6.599,-179.9457,0.0017,-1239.7284
C00696=31.947,-94.737,6.598,-179.6630,0.0048,-1241.3650
C00697=29.062,-95.605,6.597,-178.7866,0.0275,-1243.0918
C00698=26.351,-96.303,6.595,-177.4464,0.0927,-1244.6970
C00699=24.167,-96.770,6.592,-175.7648,0.2484,-1245.9780
C00700=22.417,-97.071,6.585,-173.8031,0.4429,-1246.9964
C00701=20.687,-97.336,6.576,-171.8150,0.4851,-1248.0014
C00702=18.547,-97.668,6.566,-170.1170,0.3386,-1249.2476
C00703=15.437,-98.140,6.558,-168.9780,0.1303,-1251.0609
C00704=10.884,-98.723,6.555,-168.5476,0.0211,-1253.7087
C00705=5.730,-99.155,6.555,-168.5253,-0.0014,-1256.6927
C00706=0.000,-99.321,6.555,-168.5271,0.0000,-1260.0000
C00707=0.000,-99.321,6.555,-168.5271,0.0000,-1260.0000
C00708=-5.730,-99.155,6.555,-168.5253,0.0014,-1263.3073
C00709=-10.884,-98.723,6.555,-168.5476,-0.0211,-1266.2913
C00710=-15.437,-98.140,6.558,-168.9780,-0.1303,-1268.9391
C00711=-18.547,-97.668,6.566,-170.1170,-0.3386,-1270.7524
C00712=-20.687,-97.336,6.576,-171.8150,-0.4851,-1271.9986
C00713=-22.417,-97.071,6.585,-173.8031,-0.4429,-1273.0036
C00714=-24.167,-96.770,6.592,-175.7648,-0.2484,-1274.0220
C00715=-26.351,-96.303,6.595,-177.4464,-0.0927,-1275.3030
C00716=-29.062,-95.605,6.597,-178.7866,-0.0275,-1276.9082
C00717=-31.947,-94.737,6.598,-179.6630,-0.0048,-1278.6350
C00718=-34.646,-93.803,6.599,-179.9457,-0.0017,-1280.2716
C00719=-37.090,-92.867,6.600,-179.9947,-0.0021,-1281.7712
C00720=-39.440,-91.893,6.600,-179.9947,-0.0023,-1283.2288
C00721=-41.830,-90.827,6.599,-179.9436,-0.0008,-1284.7282
C00722=-44.399,-89.579,6.598,-179.6644,0.0063,-1286.3649
C00723=-47.053,-88.152,6.597,-178.7893,0.0293,-1288.0920
C00724=-49.464,-86.729,6.595,-177.4408,0.0910,-1289.6973
C00725=-51.338,-85.515,6.592,-175.7651,0.2472,-1290.9780
C00726=-52.788,-84.491,6.585,-173.8020,0.4415,-1291.9962
C00727=-54.199,-83.455,6.576,-171.8109,0.4845,-1293.0013
C00728=-55.947,-82.176,6.566,-170.1166,0.3384,-1294.2478
C00729=-58.480,-80.311,6.558,-168.9774,0.1342,-1296.0610
C00730=-62.112,-77.504,6.555,-168.5500,0.0193,-1298.7088
C00731=-66.061,-74.165,6.555,-168.5237,-0.0027,-1301.6924
C00732=-70.230,-70.230,6.555,-168.5306,0.0000,-1305.0000
C00733=-74.165,-66.061,6.555,-168.5237,0.0027,-1308.3076
C00734=-77.504,-62.112,6.555,-168.5500,-0.0193,-1311.2912
C00735=-80.311,-58.480,6.558,-168.9774,-0.1342,-1313.9390
C00736=-82.176,-55.947,6.566,-170.1166,-0.3384,-1315.7522
C00737=-83.455,-54.199,6.576,-171.8109,-0.4845,-1316.9987
C00738=-84.491,-52.788,6.585,-173.8020,-0.4415,-1318.0038
C00739=-85.515,-51.338,6.592,-175.7651,-0.2472,-1319.0220
C00740=-86.729,-49.464,6.595,-177.4408,-0.0910,-1320.3027
C00741=-88.152,-47.053,6.597,-178.7893,-0.0293,-1321.9080
C00742=-89.579,-44.399,6.598,-179.6644,-0.0063,-1323.6351
C00743=-90.827,-41.830,6.599,-179.9436,0.0008,-1325.2718
C00744=-91.893,-39.440,6.600,-179.9947,0.0023,-1326.7712
C00745=-92.867,-37.090,6.600,-179.9947,0.0021,-1328.2288
C00746=-93.803,-34.646,6.599,-179.9457,0.0017,-1329.7284
C00747=-94.737,-31.947,6.598,-179.6630,0.0048,-1331.3650
C00748=-95.605,-29.062,6.597,-178.7866,0.0275,-1333.0918
C00749=-96.303,-26.351,6.595,-177.4464,0.0927,-1334.6970
C00750=-96.770,-24.167,6.592,-175.7648,0.2484,-1335.9780
C00751=-97.071,-22.417,6.585,-173.8031,0.4429,-1336.9964
C00752=-97.336,-20.687,6.576,-171.8150,0.4851,-1338.0014
C00753=-97.668,-18.547,6.566,-170.1170,0.3386,-1339.2476
C00754=-98.140,-15.437,6.558,-168.9780,0.1303,-1341.0609
C00755=-98.723,-10.884,6.555,-168.5476,0.0211,-1343.7087
C00756=-99.155,-5.730,6.555,-168.5253,-0.0014,-1346.6927
C00757=-99.321,0.000,6.555,-168.5271,-0.0000,-1350.0000
C00758=-99.155,5.730,6.555,-168.5253,0.0014,-1353.3073
C00759=-98.723,10.884,6.555,-168.5476,-0.0211,-1356.2913
C00760=-98.140,15.437,6.558,-168.9780,-0.1303,-1358.9391
C00761=-97.668,18.547,6.566,-170.1170,-0.3386,-1360.7524
C00762=-97.336,20.687,6.576,-171.8150,-0.4851,-1361.9986
C00763=-97.071,22.417,6.585,-173.8031,-0.4429,-1363.0036
C00764=-96.770,24.167,6.592,-175.7648,-0.2484,-1364.0220
C00765=-96.303,26.351,6.595,-177.4464,-0.0927,-1365.3030
C00766=-95.605,29.062,6.597,-178.7866,-0.0275,-1366.9082
C00767=-94.737,31.947,6.598,-179.6630,-0.0048,-1368.6350
C00768=-93.803,34.646,6.599,-179.9457,-0.0017,-1370.2716
C00769=-92.867,37.090,6.600,-179.9947,-0.0021,-1371.7712
C00770=-91.893,39.440,6.600,-179.9947,-0.0023,-1373.2288
C00771=-90.827,41.830,6.599,-179.9436,-0.0008,-1374.7282
C00772=-89.579,44.399,6.598,-179.6644,0.0063,-1376.3649
C00773=-88.152,47.053,6.597,-178.7893,0.0293,-1378.0920
C00774=-86.729,49.464,6.595,-177.4408,0.0910,-1379.6973
C00775=-85.515,51.338,6.592,-175.7651,0.2472,-1380.9780
C00776=-84.491,52.788,6.585,-173.8020,0.4415,-1381.9962
C00777=-83.455,54.199,6.576,-171.8109,0.4845,-1383.0013
C00778=-82.176,55.947,6.566,-170.1166,0.3384,-1384.2478
C00779=-80.311,58.480,6.558,-168.9774,0.1342,-1386.0610
C00780=-77.504,62.112,6.555,-168.5500,0.0193,-1388.7088
C00781=-74.165,66.061,6.555,-168.5237,-0.0027,-1391.6924
C00782=-70.230,70.230,6.555,-168.5306,0.0000,-1395.0000
C00783=-66.061,74.165,6.555,-168.5237,0.0027,-1398.3076
C00784=-62.112,77.504,6.555,-168.5500,-0.0193,-1401.2912
C00785=-58.480,80.311,6.558,-168.9774,-0.1342,-1403.9390
C00786=-55.947,82.176,6.566,-170.1166,-0.3384,-1405.7522
C00787=-54.199,83.455,6.576,-171.8109,-0.4845,-1406.9987
C00788=-52.788,84.491,6.585,-173.8020,-0.4415,-1408.0038
C00789=-51.338,85.515,6.592,-175.7651,-0.2472,-1409.0220
C00790=-49.464,86.729,6.595,-177.4408,-0.0910,-1410.3027
C00791=-47.053,88.152,6.597,-178.7893,-0.0293,-1411.9080
C00792=-44.399,89.579,6.598,-179.6644,-0.0063,-1413.6351
C00793=-41.830,90.827,6.599,-179.9436,0.0008,-1415.2718
C00794=-39.440,91.893,6.600,-179.9947,0.0023,-1416.7712
C00795=-37.090,92.867,6.600,-179.9947,0.0021,-1418.2288
C00796=-34.646,93.803,6.599,-179.9457,0.0017,-1419.7284
C00797=-31.947,94.737,6.598,-179.6630,0.0048,-1421.3650
C00798=-29.062,95.605,6.597,-178.7866,0.0275,-1423.0918
C00799=-26.351,96.303,6.595,-177.4464,0.0927,-1424.6970
C00800=-24.167,96.770,6.592,-175.7648,0.2484,-1425.9780
C00801=-22.417,97.071,6.585,-173.8031,0.4429,-1426.9964
C00802=-20.687,97.336,6.576,-171.8150,0.4851,-1428.0014
C00803=-18.547,97.668,6.566,-170.1170,0.3386,-1429.2476
C00804=-15.437,98.140,6.558,-168.9780,0.1303,-1431.0609
C00805=-10.884,98.723,6.555,-168.5476,0.0211,-1433.7087
C00806=-5.730,99.155,6.555,-168.5253,-0.0014,-1436.6927
C00807=0.000,99.321,6.555,-168.5271,0.0000,-1440.0000
C00808=0.000,98.820,8.697,-165.2384,0.0000,-1440.0000
C00809=5.684,98.656,8.697,-165.2312,0.0081,-1443.2974
C00810=10.807,98.229,8.698,-165.2649,-0.0426,-1446.2783
C00811=15.344,97.668,8.705,-165.8135,-0.3013,-1448.9284
C00812=18.436,97.247,8.723,-167.3025,-0.7735,-1450.7347
C00813=20.563,96.991,8.745,-169.5499,-1.0965,-1451.9700
C00814=22.286,96.814,8.767,-172.1574,-0.9915,-1452.9633
C00815=24.029,96.606,8.782,-174.6676,-0.5533,-1453.9678
C00816=26.202,96.222,8.789,-176.7876,-0.2036,-1455.2327
C00817=28.922,95.588,8.792,-178.4919,-0.0612,-1456.8342
C00818=31.837,94.757,8.795,-179.5978,-0.0082,-1458.5716
C00819=34.577,93.826,8.798,-179.9329,-0.0003,-1460.2300
C00820=37.066,92.876,8.800,-179.9926,0.0032,-1461.7565
C00821=39.463,91.883,8.800,-179.9925,0.0030,-1463.2431
C00822=41.895,90.794,8.798,-179.9308,-0.0004,-1464.7700
C00823=44.491,89.515,8.795,-179.5977,0.0112,-1466.4284
C00824=47.140,88.042,8.792,-178.4936,0.0579,-1468.1658
C00825=49.511,86.567,8.789,-176.7866,0.2031,-1469.7669
C00826=51.320,85.302,8.782,-174.6675,0.5502,-1471.0323
C00827=52.699,84.217,8.767,-172.1605,0.9932,-1472.0364
C00828=54.043,83.124,8.745,-169.5494,1.0947,-1473.0299
C00829=55.728,81.800,8.723,-167.3050,0.7728,-1474.2655
C00830=58.212,79.911,8.705,-165.8138,0.2999,-1476.0719
C00831=61.817,77.101,8.698,-165.2633,0.0439,-1478.7215
C00832=65.741,73.780,8.697,-165.2319,-0.0068,-1481.7023
C00833=69.877,69.877,8.697,-165.2361,0.0000,-1485.0000
C00834=73.780,65.741,8.697,-165.2319,0.0068,-1488.2977
C00835=77.101,61.817,8.698,-165.2633,-0.0439,-1491.2785
C00836=79.911,58.212,8.705,-165.8138,-0.2999,-1493.9281
C00837=81.800,55.728,8.723,-167.3050,-0.7728,-1495.7345
C00838=83.124,54.043,8.745,-169.5494,-1.0947,-1496.9701
C00839=84.217,52.699,8.767,-172.1605,-0.9932,-1497.9636
C00840=85.302,51.320,8.782,-174.6675,-0.5502,-1498.9677
C00841=86.567,49.511,8.789,-176.7866,-0.2031,-1500.2331
C00842=88.042,47.140,8.792,-178.4936,-0.0579,-1501.8342
C00843=89.515,44.491,8.795,-179.5977,-0.0112,-1503.5716
C00844=90.794,41.895,8.798,-179.9308,0.0004,-1505.2300
C00845=91.883,39.463,8.800,-179.9925,-0.0030,-1506.7569
C00846=92.876,37.066,8.800,-179.9926,-0.0032,-1508.2435
C00847=93.826,34.577,8.798,-179.9329,0.0003,-1509.7700
C00848=94.757,31.837,8.795,-179.5978,0.0082,-1511.4284
C00849=95.588,28.922,8.792,-178.4919,0.0612,-1513.1658
C00850=96.222,26.202,8.789,-176.7876,0.2036,-1514.7673
C00851=96.606,24.029,8.782,-174.6676,0.5533,-1516.0322
C00852=96.814,22.286,8.767,-172.1574,0.9915,-1517.0367
C00853=96.991,20.563,8.745,-169.5499,1.0965,-1518.0300
C00854=97.247,18.436,8.723,-167.3025,0.7735,-1519.2653
C00855=97.668,15.344,8.705,-165.8135,0.3013,-1521.0716
C00856=98.229,10.807,8.698,-165.2649,0.0426,-1523.7217
C00857=98.656,5.684,8.697,-165.2312,-0.0081,-1526.7026
C00858=98.820,0.000,8.697,-165.2384,-0.0000,-1530.0000
C00859=98.656,-5.684,8.697,-165.2312,0.0081,-1533.2974
C00860=98.229,-10.807,8.698,-165.2649,-0.0426,-1536.2783
C00861=97.668,-15.344,8.705,-165.8135,-0.3013,-1538.9284
C00862=97.247,-18.436,8.723,-167.3025,-0.7735,-1540.7347
C00863=96.991,-20.563,8.745,-169.5499,-1.0965,-1541.9700
C00864=96.814,-22.286,8.767,-172.1574,-0.9915,-1542.9633
C00865=96.606,-24.029,8.782,-174.6676,-0.5533,-1543.9678
C00866=96.222,-26.202,8.789,-176.7876,-0.2036,-1545.2327
C00867=95.588,-28.922,8.792,-178.4919,-0.0612,-1546.8342
C00868=94.757,-31.837,8.795,-179.5978,-0.0082,-1548.5716
C00869=93.826,-34.577,8.798,-179.9329,-0.0003,-1550.2300
C00870=92.876,-37.066,8.800,-179.9926,0.0032,-1551.7565
C00871=91.883,-39.463,8.800,-179.9925,0.0030,-1553.2431
C00872=90.794,-41.895,8.798,-179.9308,-0.0004,-1554.7700
C00873=89.515,-44.491,8.795,-179.5977,0.0112,-1556.4284
C00874=88.042,-47.140,8.792,-178.4936,0.0579,-1558.1658
C00875=86.567,-49.511,8.789,-176.7866,0.2031,-1559.7669
C00876=85.302,-51.320,8.782,-174.6675,0.5502,-1561.0323
C00877=84.217,-52.699,8.767,-172.1605,0.9932,-1562.0364
C00878=83.124,-54.043,8.745,-169.5494,1.0947,-1563.0299
C00879=81.800,-55.728,8.723,-167.3050,0.7728,-1564.2655
C00880=79.911,-58.212,8.705,-165.8138,0.2999,-1566.0719
C00881=77.101,-61.817,8.698,-165.2633,0.0439,-1568.7215
C00882=73.780,-65.741,8.697,-165.2319,-0.0068,-1571.7023
C00883=69.877,-69.877,8.697,-165.2361,0.0000,-1575.0000
C00884=65.741,-73.780,8.697,-165.2319,0.0068,-1578.2977
C00885=61.817,-77.101,8.698,-165.2633,-0.0439,-1581.2785
C00886=58.212,-79.911,8.705,-165.8138,-0.2999,-1583.9281
C00887=55.728,-81.800,8.723,-167.3050,-0.7728,-1585.7345
C00888=54.043,-83.124,8.745,-169.5494,-1.0947,-1586.9701
C00889=52.699,-84.217,8.767,-172.1605,-0.9932,-1587.9636
C00890=51.320,-85.302,8.782,-174.6675,-0.5502,-1588.9677
C00891=49.511,-86.567,8.789,-176.7866,-0.2031,-1590.2331
C00892=47.140,-88.042,8.792,-178.4936,-0.0579,-1591.8342
C00893=44.491,-89.515,8.795,-179.5977,-0.0112,-1593.5716
C00894=41.895,-90.794,8.798,-179.9308,0.0004,-1595.2300
C00895=39.463,-91.883,8.800,-179.9925,-0.0030,-1596.7569
C00896=37.066,-92.876,8.800,-179.9926,-0.0032,-1598.2435
C00897=34.577,-93.826,8.798,-179.9329,0.0003,-1599.7700
C00898=31.837,-94.757,8.795,-179.5978,0.0082,-1601.4284
C00899=28.922,-95.588,8.792,-178.4919,0.0612,-1603.1658
C00900=26.202,-96.222,8.789,-176.7876,0.2036,-1604.7673
C00901=24.029,-96.606,8.782,-174.6676,0.5533,-1606.0322
C00902=22.286,-96.814,8.767,-172.1574,0.9915,-1607.0367
C00903=20.563,-96.991,8.745,-169.5499,1.0965,-1608.0300
C00904=18.436,-97.247,8.723,-167.3025,0.7735,-1609.2653
C00905=15.344,-97.668,8.705,-165.8135,0.3013,-1611.0716
C00906=10.807,-98.229,8.698,-165.2649,0.0426,-1613.7217
C00907=5.684,-98.656,8.697,-165.2312,-0.0081,-1616.7026
C00908=0.000,-98.820,8.697,-165.2384,0.0000,-1620.0000
C00909=0.000,-98.820,8.697,-165.2384,0.0000,-1620.0000
C00910=-5.684,-98.656,8.697,-165.2312,0.0081,-1623.2974
C00911=-10.807,-98.229,8.698,-165.2649,-0.0426,-1626.2783
C00912=-15.344,-97.668,8.705,-165.8135,-0.3013,-1628.9284
C00913=-18.436,-97.247,8.723,-167.3025,-0.7735,-1630.7347
C00914=-20.563,-96.991,8.745,-169.5499,-1.0965,-1631.9700
C00915=-22.286,-96.814,8.767,-172.1574,-0.9915,-1632.9633
C00916=-24.029,-96.606,8.782,-174.6676,-0.5533,-1633.9678
C00917=-26.202,-96.222,8.789,-176.7876,-0.2036,-1635.2327
C00918=-28.922,-95.588,8.792,-178.4919,-0.0612,-1636.8342
C00919=-31.837,-94.757,8.795,-179.5978,-0.0082,-1638.5716
C00920=-34.577,-93.826,8.798,-179.9329,-0.0003,-1640.2300
C00921=-37.066,-92.876,8.800,-179.9926,0.0032,-1641.7565
C00922=-39.463,-91.883,8.800,-179.9925,0.0030,-1643.2431
C00923=-41.895,-90.794,8.798,-179.9308,-0.0004,-1644.7700
C00924=-44.491,-89.515,8.795,-179.5977,0.0112,-1646.4284
C00925=-47.140,-88.042,8.792,-178.4936,0.0579,-1648.1658
C00926=-49.511,-86.567,8.789,-176.7866,0.2031,-1649.7669
C00927=-51.320,-85.302,8.782,-174.6675,0.5502,-1651.0323
C00928=-52.699,-84.217,8.767,-172.1605,0.9932,-1652.0364
C00929=-54.043,-83.124,8.745,-169.5494,1.0947,-1653.0299
C00930=-55.728,-81.800,8.723,-167.3050,0.7728,-1654.2655
C00931=-58.212,-79.911,8.705,-165.8138,0.2999,-1656.0719
C00932=-61.817,-77.101,8.698,-165.2633,0.0439,-1658.7215
C00933=-65.741,-73.780,8.697,-165.2319,-0.0068,-1661.7023
C00934=-69.877,-69.877,8.697,-165.2361,0.0000,-1665.0000
C00935=-73.780,-65.741,8.697,-165.2319,0.0068,-1668.2977
C00936=-77.101,-61.817,8.698,-165.2633,-0.0439,-1671.2785
C00937=-79.911,-58.212,8.705,-165.8138,-0.2999,-1673.9281
C00938=-81.800,-55.728,8.723,-167.3050,-0.7728,-1675.7345
C00939=-83.124,-54.043,8.745,-169.5494,-1.0947,-1676.9701
C00940=-84.217,-52.699,8.767,-172.1605,-0.9932,-1677.9636
C00941=-85.302,-51.320,8.782,-174.6675,-0.5502,-1678.9677
C00942=-86.567,-49.511,8.789,-176.7866,-0.2031,-1680.2331
C00943=-88.042,-47.140,8.792,-178.4936,-0.0579,-1681.8342
C00944=-89.515,-44.491,8.795,-179.5977,-0.0112,-1683.5716
C00945=-90.794,-41.895,8.798,-179.9308,0.0004,-1685.2300
C00946=-91.883,-39.463,8.800,-179.9925,-0.0030,-1686.7569
C00947=-92.876,-37.066,8.800,-179.9926,-0.0032,-1688.2435
C00948=-93.826,-34.577,8.798,-179.9329,0.0003,-1689.7700
C00949=-94.757,-31.837,8.795,-179.5978,0.0082,-1691.4284
C00950=-95.588,-28.922,8.792,-178.4919,0.0612,-1693.1658
C00951=-96.222,-26.202,8.789,-176.7876,0.2036,-1694.7673
C00952=-96.606,-24.029,8.782,-174.6676,0.5533,-1696.0322
C00953=-96.814,-22.286,8.767,-172.1574,0.9915,-1697.0367
C00954=-96.991,-20.563,8.745,-169.5499,1.0965,-1698.0300
C00955=-97.247,-18.436,8.723,-167.3025,0.7735,-1699.2653
C00956=-97.668,-15.344,8.705,-165.8135,0.3013,-1701.0716
C00957=-98.229,-10.807,8.698,-165.2649,0.0426,-1703.7217
C00958=-98.656,-5.684,8.697,-165.2312,-0.0081,-1706.7026
C00959=-98.820,0.000,8.697,-165.2384,-0.0000,-1710.0000
C00960=-98.656,5.684,8.697,-165.2312,0.0081,-1713.2974
C00961=-98.229,10.807,8.698,-165.2649,-0.0426,-1716.2783
C00962=-97.668,15.344,8.705,-165.8135,-0.3013,-1718.9284
C00963=-97.247,18.436,8.723,-167.3025,-0.7735,-1720.7347
C00964=-96.991,20.563,8.745,-169.5499,-1.0965,-1721.9700
C00965=-96.814,22.286,8.767,-172.1574,-0.9915,-1722.9633
C00966=-96.606,24.029,8.782,-174.6676,-0.5533,-1723.9678
C00967=-96.222,26.202,8.789,-176.7876,-0.2036,-1725.2327
C00968=-95.588,28.922,8.792,-178.4919,-0.0612,-1726.8342
C00969=-94.757,31.837,8.795,-179.5978,-0.0082,-1728.5716
C00970=-93.826,34.577,8.798,-179.9329,-0.0003,-1730.2300
C00971=-92.876,37.066,8.800,-179.9926,0.0032,-1731.7565
C00972=-91.883,39.463,8.800,-179.9925,0.0030,-1733.2431
C00973=-90.794,41.895,8.798,-179.9308,-0.0004,-1734.7700
C00974=-89.515,44.491,8.795,-179.5977,0.0112,-1736.4284
C00975=-88.042,47.140,8.792,-178.4936,0.0579,-1738.1658
C00976=-86.567,49.511,8.789,-176.7866,0.2031,-1739.7669
C00977=-85.302,51.320,8.782,-174.6675,0.5502,-1741.0323
C00978=-84.217,52.699,8.767,-172.1605,0.9932,-1742.0364
C00979=-83.124,54.043,8.745,-169.5494,1.0947,-1743.0299
C00980=-81.800,55.728,8.723,-167.3050,0.7728,-1744.2655
C00981=-79.911,58.212,8.705,-165.8138,0.2999,-1746.0719
C00982=-77.101,61.817,8.698,-165.2633,0.0439,-1748.7215
C00983=-73.780,65.741,8.697,-165.2319,-0.0068,-1751.7023
C00984=-69.877,69.877,8.697,-165.2361,0.0000,-1755.0000
C00985=-65.741,73.780,8.697,-165.2319,0.0068,-1758.2977
C00986=-61.817,77.101,8.698,-165.2633,-0.0439,-1761.2785
C00987=-58.212,79.911,8.705,-165.8138,-0.2999,-1763.9281
C00988=-55.728,81.800,8.723,-167.3050,-0.7728,-1765.7345
C00989=-54.043,83.124,8.745,-169.5494,-1.0947,-1766.9701
C00990=-52.699,84.217,8.767,-172.1605,-0.9932,-1767.9636
C00991=-51.320,85.302,8.782,-174.6675,-0.5502,-1768.9677
C00992=-49.511,86.567,8.789,-176.7866,-0.2031,-1770.2331
C00993=-47.140,88.042,8.792,-178.4936,-0.0579,-1771.8342
C00994=-44.491,89.515,8.795,-179.5977,-0.0112,-1773.5716
C00995=-41.895,90.794,8.798,-179.9308,0.0004,-1775.2300
C00996=-39.463,91.883,8.800,-179.9925,-0.0030,-1776.7569
C00997=-37.066,92.876,8.800,-179.9926,-0.0032,-1778.2435
C00998=-34.577,93.826,8.798,-179.9329,0.0003,-1779.7700
C00999=-31.837,94.757,8.795,-179.5978,0.0082,-1781.4284
C01000=-28.922,95.588,8.792,-178.4919,0.0612,-1783.1658
C01001=-26.202,96.222,8.789,-176.7876,0.2036,-1784.7673
C01002=-24.029,96.606,8.782,-174.6676,0.5533,-1786.0322
C01003=-22.286,96.814,8.767,-172.1574,0.9915,-1787.0367
C01004=-20.563,96.991,8.745,-169.5499,1.0965,-1788.0300
C01005=-18.436,97.247,8.723,-167.3025,0.7735,-1789.2653
C01006=-15.344,97.668,8.705,-165.8135,0.3013,-1791.0716
C01007=-10.807,98.229,8.698,-165.2649,0.0426,-1793.7217
C01008=-5.684,98.656,8.697,-165.2312,-0.0081,-1796.7026
C01009=0.000,98.820,8.697,-165.2384,0.0000,-1800.0000
C01010=0.000,98.204,10.809,-162.2409,0.0000,-1800.0000
C01011=5.628,98.041,10.809,-162.2296,0.0065,-1803.2854
C01012=10.712,97.620,10.809,-162.2684,-0.0860,-1806.2621
C01013=15.229,97.084,10.823,-162.9320,-0.5631,-1808.9150
C01014=18.298,96.727,10.856,-164.7800,-1.4494,-1810.7121
C01015=20.409,96.562,10.898,-167.6303,-2.0251,-1811.9342
C01016=22.123,96.495,10.937,-170.8622,-1.8145,-1812.9128
C01017=23.856,96.400,10.965,-173.8063,-1.0042,-1813.8997
C01018=26.016,96.121,10.978,-176.2741,-0.3675,-1815.1448
C01019=28.748,95.567,10.985,-178.2782,-0.1051,-1816.7421
C01020=31.699,94.782,10.991,-179.5634,-0.0131,-1818.4921
C01021=34.490,93.854,10.996,-179.9202,0.0012,-1820.1777
C01022=37.037,92.887,11.000,-179.9926,0.0032,-1821.7387
C01023=39.492,91.870,11.000,-179.9925,0.0030,-1823.2613
C01024=41.977,90.753,10.996,-179.9232,0.0023,-1824.8225
C01025=44.606,89.436,10.991,-179.5644,0.0132,-1826.5076
C01026=47.248,87.904,10.985,-178.2764,0.1081,-1828.2578
C01027=49.571,86.364,10.978,-176.2728,0.3667,-1829.8549
C01028=51.296,85.034,10.965,-173.8059,1.0013,-1831.1001
C01029=52.589,83.875,10.937,-170.8611,1.8135,-1832.0874
C01030=53.849,82.711,10.898,-167.6353,2.0260,-1833.0661
C01031=55.458,81.334,10.856,-164.7794,1.4482,-1834.2883
C01032=57.880,79.417,10.823,-162.9314,0.5587,-1836.0850
C01033=61.453,76.603,10.809,-162.2669,0.0851,-1838.7375
C01034=65.346,73.305,10.809,-162.2300,-0.0070,-1841.7146
C01035=69.440,69.440,10.809,-162.2384,0.0000,-1845.0000
C01036=73.305,65.346,10.809,-162.2300,0.0070,-1848.2854
C01037=76.603,61.453,10.809,-162.2669,-0.0851,-1851.2625
C01038=79.417,57.880,10.823,-162.9314,-0.5587,-1853.9150
C01039=81.334,55.458,10.856,-164.7794,-1.4482,-1855.7117
C01040=82.711,53.849,10.898,-167.6353,-2.0260,-1856.9339
C01041=83.875,52.589,10.937,-170.8611,-1.8135,-1857.9126
C01042=85.034,51.296,10.965,-173.8059,-1.0013,-1858.8999
C01043=86.364,49.571,10.978,-176.2728,-0.3667,-1860.1451
C01044=87.904,47.248,10.985,-178.2764,-0.1081,-1861.7422
C01045=89.436,44.606,10.991,-179.5644,-0.0132,-1863.4924
C01046=90.753,41.977,10.996,-179.9232,-0.0023,-1865.1775
C01047=91.870,39.492,11.000,-179.9925,-0.0030,-1866.7387
C01048=92.887,37.037,11.000,-179.9926,-0.0032,-1868.2613
C01049=93.854,34.490,10.996,-179.9202,-0.0012,-1869.8223
C01050=94.782,31.699,10.991,-179.5634,0.0131,-1871.5079
C01051=95.567,28.748,10.985,-178.2782,0.1051,-1873.2579
C01052=96.121,26.016,10.978,-176.2741,0.3675,-1874.8552
C01053=96.400,23.856,10.965,-173.8063,1.0042,-1876.1003
C01054=96.495,22.123,10.937,-170.8622,1.8145,-1877.0872
C01055=96.562,20.409,10.898,-167.6303,2.0251,-1878.0658
C01056=96.727,18.298,10.856,-164.7800,1.4494,-1879.2879
C01057=97.084,15.229,10.823,-162.9320,0.5631,-1881.0850
C01058=97.620,10.712,10.809,-162.2684,0.0860,-1883.7379
C01059=98.041,5.628,10.809,-162.2296,-0.0065,-1886.7146
C01060=98.204,0.000,10.809,-162.2409,-0.0000,-1890.0000
C01061=98.041,-5.628,10.809,-162.2296,0.0065,-1893.2854
C01062=97.620,-10.712,10.809,-162.2684,-0.0860,-1896.2621
C01063=97.084,-15.229,10.823,-162.9320,-0.5631,-1898.9150
C01064=96.727,-18.298,10.856,-164.7800,-1.4494,-1900.7121
C01065=96.562,-20.409,10.898,-167.6303,-2.0251,-1901.9342
C01066=96.495,-22.123,10.937,-170.8622,-1.8145,-1902.9128
C01067=96.400,-23.856,10.965,-173.8063,-1.0042,-1903.8997
C01068=96.121,-26.016,10.978,-176.2741,-0.3675,-1905.1448
C01069=95.567,-28.748,10.985,-178.2782,-0.1051,-1906.7421
C01070=94.782,-31.699,10.991,-179.5634,-0.0131,-1908.4921
C01071=93.854,-34.490,10.996,-179.9202,0.0012,-1910.1777
C01072=92.887,-37.037,11.000,-179.9926,0.0032,-1911.7387
C01073=91.870,-39.492,11.000,-179.9925,0.0030,-1913.2613
C01074=90.753,-41.977,10.996,-179.9232,0.0023,-1914.8225
C01075=89.436,-44.606,10.991,-179.5644,0.0132,-1916.5076
C01076=87.904,-47.248,10.985,-178.2764,0.1081,-1918.2578
C01077=86.364,-49.571,10.978,-176.2728,0.3667,-1919.8549
C01078=85.034,-51.296,10.965,-173.8059,1.0013,-1921.1001
C01079=83.875,-52.589,10.937,-170.8611,1.8135,-1922.0874
C01080=82.711,-53.849,10.898,-167.6353,2.0260,-1923.0661
C01081=81.334,-55.458,10.856,-164.7794,1.4482,-1924.2883
C01082=79.417,-57.880,10.823,-162.9314,0.5587,-1926.0850
C01083=76.603,-61.453,10.809,-162.2669,0.0851,-1928.7375
C01084=73.305,-65.346,10.809,-162.2300,-0.0070,-1931.7146
C01085=69.440,-69.440,10.809,-162.2384,0.0000,-1935.0000
C01086=65.346,-73.305,10.809,-162.2300,0.0070,-1938.2854
C01087=61.453,-76.603,10.809,-162.2669,-0.0851,-1941.2625
C01088=57.880,-79.417,10.823,-162.9314,-0.5587,-1943.9150
C01089=55.458,-81.334,10.856,-164.7794,-1.4482,-1945.7117
C01090=53.849,-82.711,10.898,-167.6353,-2.0260,-1946.9339
C01091=52.589,-83.875,10.937,-170.8611,-1.8135,-1947.9126
C01092=51.296,-85.034,10.965,-173.8059,-1.0013,-1948.8999
C01093=49.571,-86.364,10.978,-176.2728,-0.3667,-1950.1451
C01094=47.248,-87.904,10.985,-178.2764,-0.1081,-1951.7422
C01095=44.606,-89.436,10.991,-179.5644,-0.0132,-1953.4924
C01096=41.977,-90.753,10.996,-179.9232,-0.0023,-1955.1775
C01097=39.492,-91.870,11.000,-179.9925,-0.0030,-1956.7387
C01098=37.037,-92.887,11.000,-179.9926,-0.0032,-1958.2613
C01099=34.490,-93.854,10.996,-179.9202,-0.0012,-1959.8223
C01100=31.699,-94.782,10.991,-179.5634,0.0131,-1961.5079
C01101=28.748,-95.567,10.985,-178.2782,0.1051,-1963.2579
C01102=26.016,-96.121,10.978,-176.2741,0.3675,-1964.8552
C01103=23.856,-96.400,10.965,-173.8063,1.0042,-1966.1003
C01104=22.123,-96.495,10.937,-170.8622,1.8145,-1967.0872
C01105=20.409,-96.562,10.898,-167.6303,2.0251,-1968.0658
C01106=18.298,-96.727,10.856,-164.7800,1.4494,-1969.2879
C01107=15.229,-97.084,10.823,-162.9320,0.5631,-1971.0850
C01108=10.712,-97.620,10.809,-162.2684,0.0860,-1973.7379
C01109=5.628,-98.041,10.809,-162.2296,-0.0065,-1976.7146
C01110=0.000,-98.204,10.809,-162.2409,-0.0000,-1980.0000
C01111=0.000,-98.204,10.809,-162.2409,-0.0000,-1980.0000
C01112=-5.628,-98.041,10.809,-162.2296,0.0065,-1983.2854
C01113=-10.712,-97.620,10.809,-162.2684,-0.0860,-1986.2621
C01114=-15.229,-97.084,10.823,-162.9320,-0.5631,-1988.9150
C01115=-18.298,-96.727,10.856,-164.7800,-1.4494,-1990.7121
C01116=-20.409,-96.562,10.898,-167.6303,-2.0251,-1991.9342
C01117=-22.123,-96.495,10.937,-170.8622,-1.8145,-1992.9128
C01118=-23.856,-96.400,10.965,-173.8063,-1.0042,-1993.8997
C01119=-26.016,-96.121,10.978,-176.2741,-0.3675,-1995.1448
C01120=-28.748,-95.567,10.985,-178.2782,-0.1051,-1996.7421
C01121=-31.699,-94.782,10.991,-179.5634,-0.0131,-1998.4921
C01122=-34.490,-93.854,10.996,-179.9202,0.0012,-2000.1777
C01123=-37.037,-92.887,11.000,-179.9926,0.0032,-2001.7387
C01124=-39.492,-91.870,11.000,-179.9925,0.0030,-2003.2613
C01125=-41.977,-90.753,10.996,-179.9232,0.0023,-2004.8225
C01126=-44.606,-89.436,10.991,-179.5644,0.0132,-2006.5076
C01127=-47.248,-87.904,10.985,-178.2764,0.1081,-2008.2578
C01128=-49.571,-86.364,10.978,-176.2728,0.3667,-2009.8549
C01129=-51.296,-85.034,10.965,-173.8059,1.0013,-2011.1001
C01130=-52.589,-83.875,10.937,-170.8611,1.8135,-2012.0874
C01131=-53.849,-82.711,10.898,-167.6353,2.0260,-2013.0661
C01132=-55.458,-81.334,10.856,-164.7794,1.4482,-2014.2883
C01133=-57.880,-79.417,10.823,-162.9314,0.5587,-2016.0850
C01134=-61.453,-76.603,10.809,-162.2669,0.0851,-2018.7375
C01135=-65.346,-73.305,10.809,-162.2300,-0.0070,-2021.7146
C01136=-69.440,-69.440,10.809,-162.2384,0.0000,-2025.0000
C01137=-73.305,-65.346,10.809,-162.2300,0.0070,-2028.2854
C01138=-76.603,-61.453,10.809,-162.2669,-0.0851,-2031.2625
C01139=-79.417,-57.880,10.823,-162.9314,-0.5587,-2033.9150
C01140=-81.334,-55.458,10.856,-164.7794,-1.4482,-2035.7117
C01141=-82.711,-53.849,10.898,-167.6353,-2.0260,-2036.9339
C01142=-83.875,-52.589,10.937,-170.8611,-1.8135,-2037.9126
C01143=-85.034,-51.296,10.965,-173.8059,-1.0013,-2038.8999
C01144=-86.364,-49.571,10.978,-176.2728,-0.3667,-2040.1451
C01145=-87.904,-47.248,10.985,-178.2764,-0.1081,-2041.7422
C01146=-89.436,-44.606,10.991,-179.5644,-0.0132,-2043.4924
C01147=-90.753,-41.977,10.996,-179.9232,-0.0023,-2045.1775
C01148=-91.870,-39.492,11.000,-179.9925,-0.0030,-2046.7387
C01149=-92.887,-37.037,11.000,-179.9926,-0.0032,-2048.2613
C01150=-93.854,-34.490,10.996,-179.9202,-0.0012,-2049.8223
C01151=-94.782,-31.699,10.991,-179.5634,0.0131,-2051.5079
C01152=-95.567,-28.748,10.985,-178.2782,0.1051,-2053.2579
C01153=-96.121,-26.016,10.978,-176.2741,0.3675,-2054.8552
C01154=-96.400,-23.856,10.965,-173.8063,1.0042,-2056.1003
C01155=-96.495,-22.123,10.937,-170.8622,1.8145,-2057.0872
C01156=-96.562,-20.409,10.898,-167.6303,2.0251,-2058.0658
C01157=-96.727,-18.298,10.856,-164.7800,1.4494,-2059.2879
C01158=-97.084,-15.229,10.823,-162.9320,0.5631,-2061.0850
C01159=-97.620,-10.712,10.809,-162.2684,0.0860,-2063.7379
C01160=-98.041,-5.628,10.809,-162.2296,-0.0065,-2066.7146
C01161=-98.204,0.000,10.809,-162.2409,0.0000,-2070.0000
C01162=-98.041,5.628,10.809,-162.2296,0.0065,-2073.2854
C01163=-97.620,10.712,10.809,-162.2684,-0.0860,-2076.2621
C01164=-97.084,15.229,10.823,-162.9320,-0.5631,-2078.9150
C01165=-96.727,18.298,10.856,-164.7800,-1.4494,-2080.7121
C01166=-96.562,20.409,10.898,-167.6303,-2.0251,-2081.9342
C01167=-96.495,22.123,10.937,-170.8622,-1.8145,-2082.9128
C01168=-96.400,23.856,10.965,-173.8063,-1.0042,-2083.8997
C01169=-96.121,26.016,10.978,-176.2741,-0.3675,-2085.1448
C01170=-95.567,28.748,10.985,-178.2782,-0.1051,-2086.7421
C01171=-94.782,31.699,10.991,-179.5634,-0.0131,-2088.4921
C01172=-93.854,34.490,10.996,-179.9202,0.0012,-2090.1777
C01173=-92.887,37.037,11.000,-179.9926,0.0032,-2091.7387
C01174=-91.870,39.492,11.000,-179.9925,0.0030,-2093.2613
C01175=-90.753,41.977,10.996,-179.9232,0.0023,-2094.8225
C01176=-89.436,44.606,10.991,-179.5644,0.0132,-2096.5076
C01177=-87.904,47.248,10.985,-178.2764,0.1081,-2098.2578
C01178=-86.364,49.571,10.978,-176.2728,0.3667,-2099.8549
C01179=-85.034,51.296,10.965,-173.8059,1.0013,-2101.1001
C01180=-83.875,52.589,10.937,-170.8611,1.8135,-2102.0874
C01181=-82.711,53.849,10.898,-167.6353,2.0260,-2103.0661
C01182=-81.334,55.458,10.856,-164.7794,1.4482,-2104.2883
C01183=-79.417,57.880,10.823,-162.9314,0.5587,-2106.0850
C01184=-76.603,61.453,10.809,-162.2669,0.0851,-2108.7375
C01185=-73.305,65.346,10.809,-162.2300,-0.0070,-2111.7146
C01186=-69.440,69.440,10.809,-162.2384,-0.0000,-2115.0000
C01187=-65.346,73.305,10.809,-162.2300,0.0070,-2118.2854
C01188=-61.453,76.603,10.809,-162.2669,-0.0851,-2121.2625
C01189=-57.880,79.417,10.823,-162.9314,-0.5587,-2123.9150
C01190=-55.458,81.334,10.856,-164.7794,-1.4482,-2125.7117
C01191=-53.849,82.711,10.898,-167.6353,-2.0260,-2126.9339
C01192=-52.589,83.875,10.937,-170.8611,-1.8135,-2127.9126
C01193=-51.296,85.034,10.965,-173.8059,-1.0013,-2128.8999
C01194=-49.571,86.364,10.978,-176.2728,-0.3667,-2130.1451
C01195=-47.248,87.904,10.985,-178.2764,-0.1081,-2131.7422
C01196=-44.606,89.436,10.991,-179.5644,-0.0132,-2133.4924
C01197=-41.977,90.753,10.996,-179.9232,-0.0023,-2135.1775
C01198=-39.492,91.870,11.000,-179.9925,-0.0030,-2136.7387
C01199=-37.037,92.887,11.000,-179.9926,-0.0032,-2138.2613
C01200=-34.490,93.854,10.996,-179.9202,-0.0012,-2139.8223
C01201=-31.699,94.782,10.991,-179.5634,0.0131,-2141.5079
C01202=-28.748,95.567,10.985,-178.2782,0.1051,-2143.2579
C01203=-26.016,96.121,10.978,-176.2741,0.3675,-2144.8552
C01204=-23.856,96.400,10.965,-173.8063,1.0042,-2146.1003
C01205=-22.123,96.495,10.937,-170.8622,1.8145,-2147.0872
C01206=-20.409,96.562,10.898,-167.6303,2.0251,-2148.0658
C01207=-18.298,96.727,10.856,-164.7800,1.4494,-2149.2879
C01208=-15.229,97.084,10.823,-162.9320,0.5631,-2151.0850
C01209=-10.712,97.620,10.809,-162.2684,0.0860,-2153.7379
C01210=-5.628,98.041,10.809,-162.2296,-0.0065,-2156.7146
C01211=0.000,98.204,10.809,-162.2409,0.0000,-2160.0000
C01212=0.000,97.482,12.888,-159.5244,0.0000,-2160.0000
C01213=5.562,97.322,12.887,-159.5146,0.0141,-2163.2709
C01214=10.602,96.908,12.888,-159.5595,-0.1402,-2166.2435
C01215=15.094,96.401,12.910,-160.3330,-0.9271,-2168.8988
C01216=18.135,96.115,12.963,-162.5922,-2.3851,-2170.6850
C01217=20.227,96.057,13.031,-166.1511,-3.2788,-2171.8912
C01218=21.929,96.117,13.096,-170.0088,-2.8681,-2172.8520
C01219=23.652,96.157,13.142,-173.2418,-1.5865,-2173.8189
C01220=25.795,96.000,13.164,-175.9147,-0.5761,-2175.0400
C01221=28.540,95.542,13.175,-178.1402,-0.1609,-2176.6318
C01222=31.535,94.812,13.184,-179.5543,-0.0215,-2178.3974
C01223=34.387,93.888,13.193,-179.9202,0.0013,-2180.1155
C01224=37.002,92.901,13.199,-179.9872,0.0011,-2181.7171
C01225=39.526,91.855,13.199,-179.9872,0.0007,-2183.2826
C01226=42.074,90.704,13.193,-179.9180,-0.0002,-2184.8847
C01227=44.743,89.341,13.184,-179.5541,0.0202,-2186.6022
C01228=47.377,87.740,13.175,-178.1411,0.1621,-2188.3677
C01229=49.643,86.123,13.164,-175.9142,0.5781,-2189.9600
C01230=51.269,84.717,13.142,-173.2430,1.5853,-2191.1815
C01231=52.459,83.471,13.096,-170.0061,2.8714,-2192.1481
C01232=53.620,82.225,13.031,-166.1474,3.2791,-2193.1089
C01233=55.140,80.787,12.963,-162.5898,2.3896,-2194.3149
C01234=57.492,78.839,12.910,-160.3324,0.9285,-2196.1008
C01235=61.028,76.021,12.888,-159.5593,0.1396,-2198.7567
C01236=64.884,72.750,12.887,-159.5157,-0.0113,-2201.7290
C01237=68.930,68.930,12.888,-159.5279,0.0000,-2205.0000
C01238=72.750,64.884,12.887,-159.5157,0.0113,-2208.2710
C01239=76.021,61.028,12.888,-159.5593,-0.1396,-2211.2433
C01240=78.839,57.492,12.910,-160.3324,-0.9285,-2213.8992
C01241=80.787,55.140,12.963,-162.5898,-2.3896,-2215.6851
C01242=82.225,53.620,13.031,-166.1474,-3.2791,-2216.8911
C01243=83.471,52.459,13.096,-170.0061,-2.8714,-2217.8519
C01244=84.717,51.269,13.142,-173.2430,-1.5853,-2218.8185
C01245=86.123,49.643,13.164,-175.9142,-0.5781,-2220.0400
C01246=87.740,47.377,13.175,-178.1411,-0.1621,-2221.6323
C01247=89.341,44.743,13.184,-179.5541,-0.0202,-2223.3978
C01248=90.704,42.074,13.193,-179.9180,0.0002,-2225.1153
C01249=91.855,39.526,13.199,-179.9872,-0.0007,-2226.7174
C01250=92.901,37.002,13.199,-179.9872,-0.0011,-2228.2829
C01251=93.888,34.387,13.193,-179.9202,-0.0013,-2229.8845
C01252=94.812,31.535,13.184,-179.5543,0.0215,-2231.6026
C01253=95.542,28.540,13.175,-178.1402,0.1609,-2233.3682
C01254=96.000,25.795,13.164,-175.9147,0.5761,-2234.9600
C01255=96.157,23.652,13.142,-173.2418,1.5865,-2236.1811
C01256=96.117,21.929,13.096,-170.0088,2.8681,-2237.1480
C01257=96.057,20.227,13.031,-166.1511,3.2788,-2238.1088
C01258=96.115,18.135,12.963,-162.5922,2.3851,-2239.3150
C01259=96.401,15.094,12.910,-160.3330,0.9271,-2241.1012
C01260=96.908,10.602,12.888,-159.5595,0.1402,-2243.7565
C01261=97.322,5.562,12.887,-159.5146,-0.0141,-2246.7291
C01262=97.482,0.000,12.888,-159.5244,-0.0000,-2250.0000
C01263=97.322,-5.562,12.887,-159.5146,0.0141,-2253.2709
C01264=96.908,-10.602,12.888,-159.5595,-0.1402,-2256.2435
C01265=96.401,-15.094,12.910,-160.3330,-0.9271,-2258.8988
C01266=96.115,-18.135,12.963,-162.5922,-2.3851,-2260.6850
C01267=96.057,-20.227,13.031,-166.1511,-3.2788,-2261.8912
C01268=96.117,-21.929,13.096,-170.0088,-2.8681,-2262.8520
C01269=96.157,-23.652,13.142,-173.2418,-1.5865,-2263.8189
C01270=96.000,-25.795,13.164,-175.9147,-0.5761,-2265.0400
C01271=95.542,-28.540,13.175,-178.1402,-0.1609,-2266.6318
C01272=94.812,-31.535,13.184,-179.5543,-0.0215,-2268.3974
C01273=93.888,-34.387,13.193,-179.9202,0.0013,-2270.1155
C01274=92.901,-37.002,13.199,-179.9872,0.0011,-2271.7171
C01275=91.855,-39.526,13.199,-179.9872,0.0007,-2273.2826
C01276=90.704,-42.074,13.193,-179.9180,-0.0002,-2274.8847
C01277=89.341,-44.743,13.184,-179.5541,0.0202,-2276.6022
C01278=87.740,-47.377,13.175,-178.1411,0.1621,-2278.3677
C01279=86.123,-49.643,13.164,-175.9142,0.5781,-2279.9600
C01280=84.717,-51.269,13.142,-173.2430,1.5853,-2281.1815
C01281=83.471,-52.459,13.096,-170.0061,2.8714,-2282.1481
C01282=82.225,-53.620,13.031,-166.1474,3.2791,-2283.1089
C01283=80.787,-55.140,12.963,-162.5898,2.3896,-2284.3149
C01284=78.839,-57.492,12.910,-160.3324,0.9285,-2286.1008
C01285=76.021,-61.028,12.888,-159.5593,0.1396,-2288.7567
C01286=72.750,-64.884,12.887,-159.5157,-0.0113,-2291.7290
C01287=68.930,-68.930,12.888,-159.5279,0.0000,-2295.0000
C01288=64.884,-72.750,12.887,-159.5157,0.0113,-2298.2710
C01289=61.028,-76.021,12.888,-159.5593,-0.1396,-2301.2433
C01290=57.492,-78.839,12.910,-160.3324,-0.9285,-2303.8992
C01291=55.140,-80.787,12.963,-162.5898,-2.3896,-2305.6851
C01292=53.620,-82.225,13.031,-166.1474,-3.2791,-2306.8911
C01293=52.459,-83.471,13.096,-170.0061,-2.8714,-2307.8519
C01294=51.269,-84.717,13.142,-173.2430,-1.5853,-2308.8185
C01295=49.643,-86.123,13.164,-175.9142,-0.5781,-2310.0400
C01296=47.377,-87.740,13.175,-178.1411,-0.1621,-2311.6323
C01297=44.743,-89.341,13.184,-179.5541,-0.0202,-2313.3978
C01298=42.074,-90.704,13.193,-179.9180,0.0002,-2315.1153
C01299=39.526,-91.855,13.199,-179.9872,-0.0007,-2316.7174
C01300=37.002,-92.901,13.199,-179.9872,-0.0011,-2318.2829
C01301=34.387,-93.888,13.193,-179.9202,-0.0013,-2319.8845
C01302=31.535,-94.812,13.184,-179.5543,0.0215,-2321.6026
C01303=28.540,-95.542,13.175,-178.1402,0.1609,-2323.3682
C01304=25.795,-96.000,13.164,-175.9147,0.5761,-2324.9600
C01305=23.652,-96.157,13.142,-173.2418,1.5865,-2326.1811
C01306=21.929,-96.117,13.096,-170.0088,2.8681,-2327.1480
C01307=20.227,-96.057,13.031,-166.1511,3.2788,-2328.1088
C01308=18.135,-96.115,12.963,-162.5922,2.3851,-2329.3150
C01309=15.094,-96.401,12.910,-160.3330,0.9271,-2331.1012
C01310=10.602,-96.908,12.888,-159.5595,0.1402,-2333.7565
C01311=5.562,-97.322,12.887,-159.5146,-0.0141,-2336.7291
C01312=0.000,-97.482,12.888,-159.5244,-0.0000,-2340.0000
C01313=0.000,-97.482,12.888,-159.5244,-0.0000,-2340.0000
C01314=-5.562,-97.322,12.887,-159.5146,0.0141,-2343.2709
C01315=-10.602,-96.908,12.888,-159.5595,-0.1402,-2346.2435
C01316=-15.094,-96.401,12.910,-160.3330,-0.9271,-2348.8988
C01317=-18.135,-96.115,12.963,-162.5922,-2.3851,-2350.6850
C01318=-20.227,-96.057,13.031,-166.1511,-3.2788,-2351.8912
C01319=-21.929,-96.117,13.096,-170.0088,-2.8681,-2352.8520
C01320=-23.652,-96.157,13.142,-173.2418,-1.5865,-2353.8189
C01321=-25.795,-96.000,13.164,-175.9147,-0.5761,-2355.0400
C01322=-28.540,-95.542,13.175,-178.1402,-0.1609,-2356.6318
C01323=-31.535,-94.812,13.184,-179.5543,-0.0215,-2358.3974
C01324=-34.387,-93.888,13.193,-179.9202,0.0013,-2360.1155
C01325=-37.002,-92.901,13.199,-179.9872,0.0011,-2361.7171
C01326=-39.526,-91.855,13.199,-179.9872,0.0007,-2363.2826
C01327=-42.074,-90.704,13.193,-179.9180,-0.0002,-2364.8847
C01328=-44.743,-89.341,13.184,-179.5541,0.0202,-2366.6022
C01329=-47.377,-87.740,13.175,-178.1411,0.1621,-2368.3677
C01330=-49.643,-86.123,13.164,-175.9142,0.5781,-2369.9600
C01331=-51.269,-84.717,13.142,-173.2430,1.5853,-2371.1815
C01332=-52.459,-83.471,13.096,-170.0061,2.8714,-2372.1481
C01333=-53.620,-82.225,13.031,-166.1474,3.2791,-2373.1089
C01334=-55.140,-80.787,12.963,-162.5898,2.3896,-2374.3149
C01335=-57.492,-78.839,12.910,-160.3324,0.9285,-2376.1008
C01336=-61.028,-76.021,12.888,-159.5593,0.1396,-2378.7567
C01337=-64.884,-72.750,12.887,-159.5157,-0.0113,-2381.7290
C01338=-68.930,-68.930,12.888,-159.5279,0.0000,-2385.0000
C01339=-72.750,-64.884,12.887,-159.5157,0.0113,-2388.2710
C01340=-76.021,-61.028,12.888,-159.5593,-0.1396,-2391.2433
C01341=-78.839,-57.492,12.910,-160.3324,-0.9285,-2393.8992
C01342=-80.787,-55.140,12.963,-162.5898,-2.3896,-2395.6851
C01343=-82.225,-53.620,13.031,-166.1474,-3.2791,-2396.8911
C01344=-83.471,-52.459,13.096,-170.0061,-2.8714,-2397.8519
C01345=-84.717,-51.269,13.142,-173.2430,-1.5853,-2398.8185
C01346=-86.123,-49.643,13.164,-175.9142,-0.5781,-2400.0400
C01347=-87.740,-47.377,13.175,-178.1411,-0.1621,-2401.6323
C01348=-89.341,-44.743,13.184,-179.5541,-0.0202,-2403.3978
C01349=-90.704,-42.074,13.193,-179.9180,0.0002,-2405.1153
C01350=-91.855,-39.526,13.199,-179.9872,-0.0007,-2406.7174
C01351=-92.901,-37.002,13.199,-179.9872,-0.0011,-2408.2829
C01352=-93.888,-34.387,13.193,-179.9202,-0.0013,-2409.8845
C01353=-94.812,-31.535,13.184,-179.5543,0.0215,-2411.6026
C01354=-95.542,-28.540,13.175,-178.1402,0.1609,-2413.3682
C01355=-96.000,-25.795,13.164,-175.9147,0.5761,-2414.9600
C01356=-96.157,-23.652,13.142,-173.2418,1.5865,-2416.1811
C01357=-96.117,-21.929,13.096,-170.0088,2.8681,-2417.1480
C01358=-96.057,-20.227,13.031,-166.1511,3.2788,-2418.1088
C01359=-96.115,-18.135,12.963,-162.5922,2.3851,-2419.3150
C01360=-96.401,-15.094,12.910,-160.3330,0.9271,-2421.1012
C01361=-96.908,-10.602,12.888,-159.5595,0.1402,-2423.7565
C01362=-97.322,-5.562,12.887,-159.5146,-0.0141,-2426.7291
C01363=-97.482,0.000,12.888,-159.5244,0.0000,-2430.0000
C01364=-97.322,5.562,12.887,-159.5146,0.0141,-2433.2709
C01365=-96.908,10.602,12.888,-159.5595,-0.1402,-2436.2435
C01366=-96.401,15.094,12.910,-160.3330,-0.9271,-2438.8988
C01367=-96.115,18.135,12.963,-162.5922,-2.3851,-2440.6850
C01368=-96.057,20.227,13.031,-166.1511,-3.2788,-2441.8912
C01369=-96.117,21.929,13.096,-170.0088,-2.8681,-2442.8520
C01370=-96.157,23.652,13.142,-173.2418,-1.5865,-2443.8189
C01371=-96.000,25.795,13.164,-175.9147,-0.5761,-2445.0400
C01372=-95.542,28.540,13.175,-178.1402,-0.1609,-2446.6318
C01373=-94.812,31.535,13.184,-179.5543,-0.0215,-2448.3974
C01374=-93.888,34.387,13.193,-179.9202,0.0013,-2450.1155
C01375=-92.901,37.002,13.199,-179.9872,0.0011,-2451.7171
C01376=-91.855,39.526,13.199,-179.9872,0.0007,-2453.2826
C01377=-90.704,42.074,13.193,-179.9180,-0.0002,-2454.8847
C01378=-89.341,44.743,13.184,-179.5541,0.0202,-2456.6022
C01379=-87.740,47.377,13.175,-178.1411,0.1621,-2458.3677
C01380=-86.123,49.643,13.164,-175.9142,0.5781,-2459.9600
C01381=-84.717,51.269,13.142,-173.2430,1.5853,-2461.1815
C01382=-83.471,52.459,13.096,-170.0061,2.8714,-2462.1481
C01383=-82.225,53.620,13.031,-166.1474,3.2791,-2463.1089
C01384=-80.787,55.140,12.963,-162.5898,2.3896,-2464.3149
C01385=-78.839,57.492,12.910,-160.3324,0.9285,-2466.1008
C01386=-76.021,61.028,12.888,-159.5593,0.1396,-2468.7567
C01387=-72.750,64.884,12.887,-159.5157,-0.0113,-2471.7290
C01388=-68.930,68.930,12.888,-159.5279,-0.0000,-2475.0000
C01389=-64.884,72.750,12.887,-159.5157,0.0113,-2478.2710
C01390=-61.028,76.021,12.888,-159.5593,-0.1396,-2481.2433
C01391=-57.492,78.839,12.910,-160.3324,-0.9285,-2483.8992
C01392=-55.140,80.787,12.963,-162.5898,-2.3896,-2485.6851
C01393=-53.620,82.225,13.031,-166.1474,-3.2791,-2486.8911
C01394=-52.459,83.471,13.096,-170.0061,-2.8714,-2487.8519
C01395=-51.269,84.717,13.142,-173.2430,-1.5853,-2488.8185
C01396=-49.643,86.123,13.164,-175.9142,-0.5781,-2490.0400
C01397=-47.377,87.740,13.175,-178.1411,-0.1621,-2491.6323
C01398=-44.743,89.341,13.184,-179.5541,-0.0202,-2493.3978
C01399=-42.074,90.704,13.193,-179.9180,0.0002,-2495.1153
C01400=-39.526,91.855,13.199,-179.9872,-0.0007,-2496.7174
C01401=-37.002,92.901,13.199,-179.9872,-0.0011,-2498.2829
C01402=-34.387,93.888,13.193,-179.9202,-0.0013,-2499.8845
C01403=-31.535,94.812,13.184,-179.5543,0.0215,-2501.6026
C01404=-28.540,95.542,13.175,-178.1402,0.1609,-2503.3682
C01405=-25.795,96.000,13.164,-175.9147,0.5761,-2504.9600
C01406=-23.652,96.157,13.142,-173.2418,1.5865,-2506.1811
C01407=-21.929,96.117,13.096,-170.0088,2.8681,-2507.1480
C01408=-20.227,96.057,13.031,-166.1511,3.2788,-2508.1088
C01409=-18.135,96.115,12.963,-162.5922,2.3851,-2509.3150
C01410=-15.094,96.401,12.910,-160.3330,0.9271,-2511.1012
C01411=-10.602,96.908,12.888,-159.5595,0.1402,-2513.7565
C01412=-5.562,97.322,12.887,-159.5146,-0.0141,-2516.7291
C01413=0.000,97.482,12.888,-159.5244,0.0000,-2520.0000
C01414=0.000,96.668,14.931,-157.0813,0.0000,-2520.0000
C01415=5.488,96.511,14.930,-157.0684,0.0174,-2523.2546
C01416=10.476,96.104,14.932,-157.1235,-0.2080,-2526.2211
C01417=14.942,95.628,14.964,-158.0076,-1.4009,-2528.8807
C01418=17.951,95.422,15.043,-160.7627,-3.6020,-2530.6541
C01419=20.020,95.481,15.144,-165.1918,-4.7929,-2531.8420
C01420=21.708,95.685,15.242,-169.6927,-4.0631,-2532.7823
C01421=23.417,95.878,15.312,-173.0314,-2.2444,-2533.7251
C01422=25.541,95.862,15.345,-175.7358,-0.8170,-2534.9190
C01423=28.302,95.513,15.362,-178.0939,-0.2242,-2536.5054
C01424=31.347,94.846,15.376,-179.5796,-0.0243,-2538.2889
C01425=34.268,93.927,15.390,-179.9148,-0.0006,-2540.0438
C01426=36.962,92.916,15.399,-179.9872,0.0011,-2541.6927
C01427=39.566,91.838,15.399,-179.9872,0.0007,-2543.3075
C01428=42.186,90.648,15.390,-179.9180,-0.0003,-2544.9564
C01429=44.901,89.232,15.376,-179.5823,0.0271,-2546.7113
C01430=47.525,87.551,15.362,-178.0923,0.2230,-2548.4943
C01431=49.724,85.845,15.345,-175.7352,0.8188,-2550.0807
C01432=51.237,84.354,15.312,-173.0353,2.2423,-2551.2747
C01433=52.309,83.010,15.242,-169.6915,4.0591,-2552.2172
C01434=53.359,81.672,15.144,-165.1895,4.7934,-2553.1579
C01435=54.780,80.167,15.043,-160.7634,3.5991,-2554.3457
C01436=57.054,78.185,14.964,-158.0062,1.3994,-2556.1194
C01437=60.548,75.364,14.932,-157.1245,0.2111,-2558.7787
C01438=64.363,72.124,14.930,-157.0694,-0.0184,-2561.7455
C01439=68.355,68.355,14.931,-157.0774,-0.0000,-2565.0000
C01440=72.124,64.363,14.930,-157.0694,0.0184,-2568.2545
C01441=75.364,60.548,14.932,-157.1245,-0.2111,-2571.2213
C01442=78.185,57.054,14.964,-158.0062,-1.3994,-2573.8806
C01443=80.167,54.780,15.043,-160.7634,-3.5991,-2575.6543
C01444=81.672,53.359,15.144,-165.1895,-4.7934,-2576.8421
C01445=83.010,52.309,15.242,-169.6915,-4.0591,-2577.7828
C01446=84.354,51.237,15.312,-173.0353,-2.2423,-2578.7253
C01447=85.845,49.724,15.345,-175.7352,-0.8188,-2579.9193
C01448=87.551,47.525,15.362,-178.0923,-0.2230,-2581.5057
C01449=89.232,44.901,15.376,-179.5823,-0.0271,-2583.2887
C01450=90.648,42.186,15.390,-179.9180,0.0003,-2585.0436
C01451=91.838,39.566,15.399,-179.9872,-0.0007,-2586.6925
C01452=92.916,36.962,15.399,-179.9872,-0.0011,-2588.3073
C01453=93.927,34.268,15.390,-179.9148,0.0006,-2589.9562
C01454=94.846,31.347,15.376,-179.5796,0.0243,-2591.7111
C01455=95.513,28.302,15.362,-178.0939,0.2242,-2593.4946
C01456=95.862,25.541,15.345,-175.7358,0.8170,-2595.0810
C01457=95.878,23.417,15.312,-173.0314,2.2444,-2596.2749
C01458=95.685,21.708,15.242,-169.6927,4.0631,-2597.2177
C01459=95.481,20.020,15.144,-165.1918,4.7929,-2598.1580
C01460=95.422,17.951,15.043,-160.7627,3.6020,-2599.3459
C01461=95.628,14.942,14.964,-158.0076,1.4009,-2601.1193
C01462=96.104,10.476,14.932,-157.1235,0.2080,-2603.7789
C01463=96.511,5.488,14.930,-157.0684,-0.0174,-2606.7454
C01464=96.668,0.000,14.931,-157.0813,-0.0000,-2610.0000
C01465=96.511,-5.488,14.930,-157.0684,0.0174,-2613.2546
C01466=96.104,-10.476,14.932,-157.1235,-0.2080,-2616.2211
C01467=95.628,-14.942,14.964,-158.0076,-1.4009,-2618.8807
C01468=95.422,-17.951,15.043,-160.7627,-3.6020,-2620.6541
C01469=95.481,-20.020,15.144,-165.1918,-4.7929,-2621.8420
C01470=95.685,-21.708,15.242,-169.6927,-4.0631,-2622.7823
C01471=95.878,-23.417,15.312,-173.0314,-2.2444,-2623.7251
C01472=95.862,-25.541,15.345,-175.7358,-0.8170,-2624.9190
C01473=95.513,-28.302,15.362,-178.0939,-0.2242,-2626.5054
C01474=94.846,-31.347,15.376,-179.5796,-0.0243,-2628.2889
C01475=93.927,-34.268,15.390,-179.9148,-0.0006,-2630.0438
C01476=92.916,-36.962,15.399,-179.9872,0.0011,-2631.6927
C01477=91.838,-39.566,15.399,-179.9872,0.0007,-2633.3075
C01478=90.648,-42.186,15.390,-179.9180,-0.0003,-2634.9564
C01479=89.232,-44.901,15.376,-179.5823,0.0271,-2636.7113
C01480=87.551,-47.525,15.362,-178.0923,0.2230,-2638.4943
C01481=85.845,-49.724,15.345,-175.7352,0.8188,-2640.0807
C01482=84.354,-51.237,15.312,-173.0353,2.2423,-2641.2747
C01483=83.010,-52.309,15.242,-169.6915,4.0591,-2642.2172
C01484=81.672,-53.359,15.144,-165.1895,4.7934,-2643.1579
C01485=80.167,-54.780,15.043,-160.7634,3.5991,-2644.3457
C01486=78.185,-57.054,14.964,-158.0062,1.3994,-2646.1194
C01487=75.364,-60.548,14.932,-157.1245,0.2111,-2648.7787
C01488=72.124,-64.363,14.930,-157.0694,-0.0184,-2651.7455
C01489=68.355,-68.355,14.931,-157.0774,0.0000,-2655.0000
C01490=64.363,-72.124,14.930,-157.0694,0.0184,-2658.2545
C01491=60.548,-75.364,14.932,-157.1245,-0.2111,-2661.2213
C01492=57.054,-78.185,14.964,-158.0062,-1.3994,-2663.8806
C01493=54.780,-80.167,15.043,-160.7634,-3.5991,-2665.6543
C01494=53.359,-81.672,15.144,-165.1895,-4.7934,-2666.8421
C01495=52.309,-83.010,15.242,-169.6915,-4.0591,-2667.7828
C01496=51.237,-84.354,15.312,-173.0353,-2.2423,-2668.7253
C01497=49.724,-85.845,15.345,-175.7352,-0.8188,-2669.9193
C01498=47.525,-87.551,15.362,-178.0923,-0.2230,-2671.5057
C01499=44.901,-89.232,15.376,-179.5823,-0.0271,-2673.2887
C01500=42.186,-90.648,15.390,-179.9180,0.0003,-2675.0436
C01501=39.566,-91.838,15.399,-179.9872,-0.0007,-2676.6925
C01502=36.962,-92.916,15.399,-179.9872,-0.0011,-2678.3073
C01503=34.268,-93.927,15.390,-179.9148,0.0006,-2679.9562
C01504=31.347,-94.846,15.376,-179.5796,0.0243,-2681.7111
C01505=28.302,-95.513,15.362,-178.0939,0.2242,-2683.4946
C01506=25.541,-95.862,15.345,-175.7358,0.8170,-2685.0810
C01507=23.417,-95.878,15.312,-173.0314,2.2444,-2686.2749
C01508=21.708,-95.685,15.242,-169.6927,4.0631,-2687.2177
C01509=20.020,-95.481,15.144,-165.1918,4.7929,-2688.1580
C01510=17.951,-95.422,15.043,-160.7627,3.6020,-2689.3459
C01511=14.942,-95.628,14.964,-158.0076,1.4009,-2691.1193
C01512=10.476,-96.104,14.932,-157.1235,0.2080,-2693.7789
C01513=5.488,-96.511,14.930,-157.0684,-0.0174,-2696.7454
C01514=0.000,-96.668,14.931,-157.0813,-0.0000,-2700.0000
C01515=0.000,-96.668,14.931,-157.0813,-0.0000,-2700.0000
C01516=-5.488,-96.511,14.930,-157.0684,0.0174,-2703.2546
C01517=-10.476,-96.104,14.932,-157.1235,-0.2080,-2706.2211
C01518=-14.942,-95.628,14.964,-158.0076,-1.4009,-2708.8807
C01519=-17.951,-95.422,15.043,-160.7627,-3.6020,-2710.6541
C01520=-20.020,-95.481,15.144,-165.1918,-4.7929,-2711.8420
C01521=-21.708,-95.685,15.242,-169.6927,-4.0631,-2712.7823
C01522=-23.417,-95.878,15.312,-173.0314,-2.2444,-2713.7251
C01523=-25.541,-95.862,15.345,-175.7358,-0.8170,-2714.9190
C01524=-28.302,-95.513,15.362,-178.0939,-0.2242,-2716.5054
C01525=-31.347,-94.846,15.376,-179.5796,-0.0243,-2718.2889
C01526=-34.268,-93.927,15.390,-179.9148,-0.0006,-2720.0438
C01527=-36.962,-92.916,15.399,-179.9872,0.0011,-2721.6927
C01528=-39.566,-91.838,15.399,-179.9872,0.0007,-2723.3075
C01529=-42.186,-90.648,15.390,-179.9180,-0.0003,-2724.9564
C01530=-44.901,-89.232,15.376,-179.5823,0.0271,-2726.7113
C01531=-47.525,-87.551,15.362,-178.0923,0.2230,-2728.4943
C01532=-49.724,-85.845,15.345,-175.7352,0.8188,-2730.0807
C01533=-51.237,-84.354,15.312,-173.0353,2.2423,-2731.2747
C01534=-52.309,-83.010,15.242,-169.6915,4.0591,-2732.2172
C01535=-53.359,-81.672,15.144,-165.1895,4.7934,-2733.1579
C01536=-54.780,-80.167,15.043,-160.7634,3.5991,-2734.3457
C01537=-57.054,-78.185,14.964,-158.0062,1.3994,-2736.1194
C01538=-60.548,-75.364,14.932,-157.1245,0.2111,-2738.7787
C01539=-64.363,-72.124,14.930,-157.0694,-0.0184,-2741.7455
C01540=-68.355,-68.355,14.931,-157.0774,0.0000,-2745.0000
C01541=-72.124,-64.363,14.930,-157.0694,0.0184,-2748.2545
C01542=-75.364,-60.548,14.932,-157.1245,-0.2111,-2751.2213
C01543=-78.185,-57.054,14.964,-158.0062,-1.3994,-2753.8806
C01544=-80.167,-54.780,15.043,-160.7634,-3.5991,-2755.6543
C01545=-81.672,-53.359,15.144,-165.1895,-4.7934,-2756.8421
C01546=-83.010,-52.309,15.242,-169.6915,-4.0591,-2757.7828
C01547=-84.354,-51.237,15.312,-173.0353,-2.2423,-2758.7253
C01548=-85.845,-49.724,15.345,-175.7352,-0.8188,-2759.9193
C01549=-87.551,-47.525,15.362,-178.0923,-0.2230,-2761.5057
C01550=-89.232,-44.901,15.376,-179.5823,-0.0271,-2763.2887
C01551=-90.648,-42.186,15.390,-179.9180,0.0003,-2765.0436
C01552=-91.838,-39.566,15.399,-179.9872,-0.0007,-2766.6925
C01553=-92.916,-36.962,15.399,-179.9872,-0.0011,-2768.3073
C01554=-93.927,-34.268,15.390,-179.9148,0.0006,-2769.9562
C01555=-94.846,-31.347,15.376,-179.5796,0.0243,-2771.7111
C01556=-95.513,-28.302,15.362,-178.0939,0.2242,-2773.4946
C01557=-95.862,-25.541,15.345,-175.7358,0.8170,-2775.0810
C01558=-95.878,-23.417,15.312,-173.0314,2.2444,-2776.2749
C01559=-95.685,-21.708,15.242,-169.6927,4.0631,-2777.2177
C01560=-95.481,-20.020,15.144,-165.1918,4.7929,-2778.1580
C01561=-95.422,-17.951,15.043,-160.7627,3.6020,-2779.3459
C01562=-95.628,-14.942,14.964,-158.0076,1.4009,-2781.1193
C01563=-96.104,-10.476,14.932,-157.1235,0.2080,-2783.7789
C01564=-96.511,-5.488,14.930,-157.0684,-0.0174,-2786.7454
C01565=-96.668,0.000,14.931,-157.0813,0.0000,-2790.0000
C01566=-96.511,5.488,14.930,-157.0684,0.0174,-2793.2546
C01567=-96.104,10.476,14.932,-157.1235,-0.2080,-2796.2211
C01568=-95.628,14.942,14.964,-158.0076,-1.4009,-2798.8807
C01569=-95.422,17.951,15.043,-160.7627,-3.6020,-2800.6541
C01570=-95.481,20.020,15.144,-165.1918,-4.7929,-2801.8420
C01571=-95.685,21.708,15.242,-169.6927,-4.0631,-2802.7823
C01572=-95.878,23.417,15.312,-173.0314,-2.2444,-2803.7251
C01573=-95.862,25.541,15.345,-175.7358,-0.8170,-2804.9190
C01574=-95.513,28.302,15.362,-178.0939,-0.2242,-2806.5054
C01575=-94.846,31.347,15.376,-179.5796,-0.0243,-2808.2889
C01576=-93.927,34.268,15.390,-179.9148,-0.0006,-2810.0438
C01577=-92.916,36.962,15.399,-179.9872,0.0011,-2811.6927
C01578=-91.838,39.566,15.399,-179.9872,0.0007,-2813.3075
C01579=-90.648,42.186,15.390,-179.9180,-0.0003,-2814.9564
C01580=-89.232,44.901,15.376,-179.5823,0.0271,-2816.7113
C01581=-87.551,47.525,15.362,-178.0923,0.2230,-2818.4943
C01582=-85.845,49.724,15.345,-175.7352,0.8188,-2820.0807
C01583=-84.354,51.237,15.312,-173.0353,2.2423,-2821.2747
C01584=-83.010,52.309,15.242,-169.6915,4.0591,-2822.2172
C01585=-81.672,53.359,15.144,-165.1895,4.7934,-2823.1579
C01586=-80.167,54.780,15.043,-160.7634,3.5991,-2824.3457
C01587=-78.185,57.054,14.964,-158.0062,1.3994,-2826.1194
C01588=-75.364,60.548,14.932,-157.1245,0.2111,-2828.7787
C01589=-72.124,64.363,14.930,-157.0694,-0.0184,-2831.7455
C01590=-68.355,68.355,14.931,-157.0774,-0.0000,-2835.0000
C01591=-64.363,72.124,14.930,-157.0694,0.0184,-2838.2545
C01592=-60.548,75.364,14.932,-157.1245,-0.2111,-2841.2213
C01593=-57.054,78.185,14.964,-158.0062,-1.3994,-2843.8806
C01594=-54.780,80.167,15.043,-160.7634,-3.5991,-2845.6543
C01595=-53.359,81.672,15.144,-165.1895,-4.7934,-2846.8421
C01596=-52.309,83.010,15.242,-169.6915,-4.0591,-2847.7828
C01597=-51.237,84.354,15.312,-173.0353,-2.2423,-2848.7253
C01598=-49.724,85.845,15.345,-175.7352,-0.8188,-2849.9193
C01599=-47.525,87.551,15.362,-178.0923,-0.2230,-2851.5057
C01600=-44.901,89.232,15.376,-179.5823,-0.0271,-2853.2887
C01601=-42.186,90.648,15.390,-179.9180,0.0003,-2855.0436
C01602=-39.566,91.838,15.399,-179.9872,-0.0007,-2856.6925
C01603=-36.962,92.916,15.399,-179.9872,-0.0011,-2858.3073
C01604=-34.268,93.927,15.390,-179.9148,0.0006,-2859.9562
C01605=-31.347,94.846,15.376,-179.5796,0.0243,-2861.7111
C01606=-28.302,95.513,15.362,-178.0939,0.2242,-2863.4946
C01607=-25.541,95.862,15.345,-175.7358,0.8170,-2865.0810
C01608=-23.417,95.878,15.312,-173.0314,2.2444,-2866.2749
C01609=-21.708,95.685,15.242,-169.6927,4.0631,-2867.2177
C01610=-20.020,95.481,15.144,-165.1918,4.7929,-2868.1580
C01611=-17.951,95.422,15.043,-160.7627,3.6020,-2869.3459
C01612=-14.942,95.628,14.964,-158.0076,1.4009,-2871.1193
C01613=-10.476,96.104,14.932,-157.1235,0.2080,-2873.7789
C01614=-5.488,96.511,14.930,-157.0684,-0.0174,-2876.7454
C01615=0.000,96.668,14.931,-157.0813,0.0000,-2880.0000
C01616=0.000,95.772,16.941,-154.8879,0.0000,-2880.0000
C01617=5.406,95.617,16.939,-154.8750,0.0274,-2883.2359
C01618=10.339,95.219,16.941,-154.9335,-0.3011,-2886.1970
C01619=14.774,94.777,16.986,-155.9417,-1.9916,-2888.8601
C01620=17.748,94.656,17.095,-159.3411,-5.0626,-2890.6197
C01621=19.790,94.842,17.237,-164.8285,-6.4355,-2891.7864
C01622=21.462,95.203,17.374,-169.9520,-5.2148,-2892.7041
C01623=23.155,95.565,17.473,-173.2181,-2.8849,-2893.6200
C01624=25.257,95.708,17.521,-175.7539,-1.0630,-2894.7831
C01625=28.035,95.481,17.545,-178.1294,-0.2806,-2896.3632
C01626=31.135,94.884,17.565,-179.6411,-0.0273,-2898.1666
C01627=34.135,93.972,17.585,-179.9202,0.0015,-2899.9634
C01628=36.917,92.934,17.598,-179.9926,0.0032,-2901.6649
C01629=39.610,91.818,17.598,-179.9925,0.0030,-2903.3352
C01630=42.311,90.585,17.585,-179.9180,-0.0004,-2905.0366
C01631=45.077,89.109,17.565,-179.6386,0.0291,-2906.8332
C01632=47.692,87.339,17.545,-178.1307,0.2787,-2908.6370
C01633=49.816,85.535,17.521,-175.7503,1.0646,-2910.2167
C01634=51.202,83.948,17.473,-173.2162,2.8847,-2911.3801
C01635=52.143,82.495,17.374,-169.9475,5.2185,-2912.2959
C01636=53.070,81.058,17.237,-164.8269,6.4371,-2913.2134
C01637=54.382,79.482,17.095,-159.3399,5.0676,-2914.3801
C01638=56.571,77.464,16.986,-155.9409,1.9875,-2916.1402
C01639=60.019,74.640,16.941,-154.9325,0.3004,-2918.8032
C01640=63.789,71.434,16.939,-154.8745,-0.0271,-2921.7642
C01641=67.721,67.721,16.941,-154.8876,-0.0000,-2925.0000
C01642=71.434,63.789,16.939,-154.8745,0.0271,-2928.2358
C01643=74.640,60.019,16.941,-154.9325,-0.3004,-2931.1968
C01644=77.464,56.571,16.986,-155.9409,-1.9875,-2933.8598
C01645=79.482,54.382,17.095,-159.3399,-5.0676,-2935.6199
C01646=81.058,53.070,17.237,-164.8269,-6.4371,-2936.7866
C01647=82.495,52.143,17.374,-169.9475,-5.2185,-2937.7041
C01648=83.948,51.202,17.473,-173.2162,-2.8847,-2938.6199
C01649=85.535,49.816,17.521,-175.7503,-1.0646,-2939.7833
C01650=87.339,47.692,17.545,-178.1307,-0.2787,-2941.3630
C01651=89.109,45.077,17.565,-179.6386,-0.0291,-2943.1668
C01652=90.585,42.311,17.585,-179.9180,0.0004,-2944.9634
C01653=91.818,39.610,17.598,-179.9925,-0.0030,-2946.6648
C01654=92.934,36.917,17.598,-179.9926,-0.0032,-2948.3351
C01655=93.972,34.135,17.585,-179.9202,-0.0015,-2950.0366
C01656=94.884,31.135,17.565,-179.6411,0.0273,-2951.8334
C01657=95.481,28.035,17.545,-178.1294,0.2806,-2953.6368
C01658=95.708,25.257,17.521,-175.7539,1.0630,-2955.2169
C01659=95.565,23.155,17.473,-173.2181,2.8849,-2956.3800
C01660=95.203,21.462,17.374,-169.9520,5.2148,-2957.2959
C01661=94.842,19.790,17.237,-164.8285,6.4355,-2958.2136
C01662=94.656,17.748,17.095,-159.3411,5.0626,-2959.3803
C01663=94.777,14.774,16.986,-155.9417,1.9916,-2961.1399
C01664=95.219,10.339,16.941,-154.9335,0.3011,-2963.8030
C01665=95.617,5.406,16.939,-154.8750,-0.0274,-2966.7641
C01666=95.772,0.000,16.941,-154.8879,0.0000,-2970.0000
C01667=95.617,-5.406,16.939,-154.8750,0.0274,-2973.2359
C01668=95.219,-10.339,16.941,-154.9335,-0.3011,-2976.1970
C01669=94.777,-14.774,16.986,-155.9409,-1.9854,-2978.8601
C01670=94.656,-17.748,17.095,-159.3411,-5.0626,-2980.6197
C01671=94.842,-19.790,17.237,-164.8285,-6.4355,-2981.7864
C01672=95.203,-21.462,17.374,-169.9520,-5.2148,-2982.7041
C01673=95.565,-23.155,17.473,-173.2181,-2.8849,-2983.6200
C01674=95.708,-25.257,17.521,-175.7539,-1.0630,-2984.7831
C01675=95.481,-28.035,17.545,-178.1294,-0.2806,-2986.3632
C01676=94.884,-31.135,17.565,-179.6411,-0.0273,-2988.1666
C01677=93.972,-34.135,17.585,-179.9202,0.0015,-2989.9634
C01678=92.934,-36.917,17.598,-179.9926,0.0032,-2991.6649
C01679=91.818,-39.610,17.598,-179.9925,0.0030,-2993.3352
C01680=90.585,-42.311,17.585,-179.9180,-0.0004,-2995.0366
C01681=89.109,-45.077,17.565,-179.6386,0.0291,-2996.8332
C01682=87.339,-47.692,17.545,-178.1307,0.2787,-2998.6370
C01683=85.535,-49.816,17.521,-175.7503,1.0646,-3000.2167
C01684=83.948,-51.202,17.473,-173.2162,2.8847,-3001.3801
C01685=82.495,-52.143,17.374,-169.9475,5.2185,-3002.2959
C01686=81.058,-53.070,17.237,-164.8269,6.4371,-3003.2134
C01687=79.482,-54.382,17.095,-159.3399,5.0676,-3004.3801
C01688=77.464,-56.571,16.986,-155.9409,1.9875,-3006.1402
C01689=74.640,-60.019,16.941,-154.9325,0.3004,-3008.8032
C01690=71.434,-63.789,16.939,-154.8745,-0.0271,-3011.7642
C01691=67.721,-67.721,16.941,-154.8876,0.0000,-3015.0000
C01692=63.789,-71.434,16.939,-154.8745,0.0271,-3018.2358
C01693=60.019,-74.640,16.941,-154.9325,-0.3004,-3021.1968
C01694=56.571,-77.464,16.986,-155.9409,-1.9875,-3023.8598
C01695=54.382,-79.482,17.095,-159.3399,-5.0676,-3025.6199
C01696=53.070,-81.058,17.237,-164.8269,-6.4371,-3026.7866
C01697=52.143,-82.495,17.374,-169.9475,-5.2185,-3027.7041
C01698=51.202,-83.948,17.473,-173.2162,-2.8847,-3028.6199
C01699=49.816,-85.535,17.521,-175.7503,-1.0646,-3029.7833
C01700=47.692,-87.339,17.545,-178.1307,-0.2787,-3031.3630
C01701=45.077,-89.109,17.565,-179.6386,-0.0291,-3033.1668
C01702=42.311,-90.585,17.585,-179.9180,0.0004,-3034.9634
C01703=39.610,-91.818,17.598,-179.9925,-0.0030,-3036.6648
C01704=36.917,-92.934,17.598,-179.9926,-0.0032,-3038.3351
C01705=34.135,-93.972,17.585,-179.9202,-0.0015,-3040.0366
C01706=31.135,-94.884,17.565,-179.6411,0.0273,-3041.8334
C01707=28.035,-95.481,17.545,-178.1294,0.2806,-3043.6368
C01708=25.257,-95.708,17.521,-175.7539,1.0630,-3045.2169
C01709=23.155,-95.565,17.473,-173.2181,2.8849,-3046.3800
C01710=21.462,-95.203,17.374,-169.9520,5.2148,-3047.2959
C01711=19.790,-94.842,17.237,-164.8285,6.4355,-3048.2136
C01712=17.748,-94.656,17.095,-159.3411,5.0626,-3049.3803
C01713=14.774,-94.777,16.986,-155.9417,1.9916,-3051.1399
C01714=10.339,-95.219,16.941,-154.9335,0.3011,-3053.8030
C01715=5.406,-95.617,16.939,-154.8750,-0.0274,-3056.7641
C01716=0.000,-95.772,16.941,-154.8879,-0.0000,-3060.0000
C01717=0.000,-95.772,16.941,-154.8879,-0.0000,-3060.0000
C01718=-5.406,-95.617,16.939,-154.8750,0.0274,-3063.2359
C01719=-10.339,-95.219,16.941,-154.9335,-0.3011,-3066.1970
C01720=-14.774,-94.777,16.986,-155.9409,-1.9854,-3068.8601
C01721=-17.748,-94.656,17.095,-159.3411,-5.0626,-3070.6197
C01722=-19.790,-94.842,17.237,-164.8285,-6.4355,-3071.7864
C01723=-21.462,-95.203,17.374,-169.9520,-5.2148,-3072.7041
C01724=-23.155,-95.565,17.473,-173.2181,-2.8849,-3073.6200
C01725=-25.257,-95.708,17.521,-175.7539,-1.0630,-3074.7831
C01726=-28.035,-95.481,17.545,-178.1294,-0.2806,-3076.3632
C01727=-31.135,-94.884,17.565,-179.6411,-0.0273,-3078.1666
C01728=-34.135,-93.972,17.585,-179.9202,0.0015,-3079.9634
C01729=-36.917,-92.934,17.598,-179.9926,0.0032,-3081.6649
C01730=-39.610,-91.818,17.598,-179.9925,0.0030,-3083.3352
C01731=-42.311,-90.585,17.585,-179.9180,-0.0004,-3085.0366
C01732=-45.077,-89.109,17.565,-179.6386,0.0291,-3086.8332
C01733=-47.692,-87.339,17.545,-178.1307,0.2787,-3088.6370
C01734=-49.816,-85.535,17.521,-175.7503,1.0646,-3090.2167
C01735=-51.202,-83.948,17.473,-173.2162,2.8847,-3091.3801
C01736=-52.143,-82.495,17.374,-169.9475,5.2185,-3092.2959
C01737=-53.070,-81.058,17.237,-164.8269,6.4371,-3093.2134
C01738=-54.382,-79.482,17.095,-159.3399,5.0676,-3094.3801
C01739=-56.571,-77.464,16.986,-155.9409,1.9875,-3096.1402
C01740=-60.019,-74.640,16.941,-154.9325,0.3004,-3098.8032
C01741=-63.789,-71.434,16.939,-154.8745,-0.0271,-3101.7642
C01742=-67.721,-67.721,16.941,-154.8876,0.0000,-3105.0000
C01743=-71.434,-63.789,16.939,-154.8745,0.0271,-3108.2358
C01744=-74.640,-60.019,16.941,-154.9325,-0.3004,-3111.1968
C01745=-77.464,-56.571,16.986,-155.9409,-1.9875,-3113.8598
C01746=-79.482,-54.382,17.095,-159.3399,-5.0676,-3115.6199
C01747=-81.058,-53.070,17.237,-164.8269,-6.4371,-3116.7866
C01748=-82.495,-52.143,17.374,-169.9475,-5.2185,-3117.7041
C01749=-83.948,-51.202,17.473,-173.2162,-2.8847,-3118.6199
C01750=-85.535,-49.816,17.521,-175.7503,-1.0646,-3119.7833
C01751=-87.339,-47.692,17.545,-178.1307,-0.2787,-3121.3630
C01752=-89.109,-45.077,17.565,-179.6386,-0.0291,-3123.1668
C01753=-90.585,-42.311,17.585,-179.9180,0.0004,-3124.9634
C01754=-91.818,-39.610,17.598,-179.9925,-0.0030,-3126.6648
C01755=-92.934,-36.917,17.598,-179.9926,-0.0032,-3128.3351
C01756=-93.972,-34.135,17.585,-179.9202,-0.0015,-3130.0366
C01757=-94.884,-31.135,17.565,-179.6411,0.0273,-3131.8334
C01758=-95.481,-28.035,17.545,-178.1294,0.2806,-3133.6368
C01759=-95.708,-25.257,17.521,-175.7539,1.0630,-3135.2169
C01760=-95.565,-23.155,17.473,-173.2181,2.8849,-3136.3800
C01761=-95.203,-21.462,17.374,-169.9520,5.2148,-3137.2959
C01762=-94.842,-19.790,17.237,-164.8285,6.4355,-3138.2136
C01763=-94.656,-17.748,17.095,-159.3411,5.0626,-3139.3803
C01764=-94.777,-14.774,16.986,-155.9417,1.9916,-3141.1399
